FUNCTION_BLOCK "FB_FW_x"   // FB11, STL
TITLE = Fahrwagensteuerung
{ S7_Optimized_Access := 'FALSE' }
AUTHOR : MS
// stored: AutoNumber false
   VAR
      ZST : Struct   // ZUSTAND
         BEREIT : Bool;   // Fahrwagen wartet auf Fahrbefehl
         AKTIV : Bool;   // Fahrwagen bearbeitet Fahrbefehl
         FEHLER : Bool;   // Fahrwagen gestört
         REFERENZIERT : Bool;   // REFERENZIERT
         HEBEN_AKT : Bool;   // Heben aktiv
         SENKEN_AKT : Bool;   // Senken aktiv
         VORWAERTS_AKT : Bool;   // Fahrt zur nächst höheren Position aktiv
         RUECKWAERTS_AKT : Bool;   // Fahrt zur nächst niedrigeren Position aktiv
         Befehl_ok : Bool;   // Befehl angenommen
         Befehl_nok : Bool;   // Befehl abgelehnt
         Befehl_done : Bool;   // Befehl ausgeführt
         Tipp : Bool;   // BA Tippbetrieb interner Zustand
         Hand : Bool;   // BA Handbetrieb interner Zustand
         Auto_Stop : Bool;   // BA Automatikbetrieb angehalten interner Zustand
         Auto : Bool;   // BA Auto interner Zustand
         Semi : Bool;   // Semiautomatik
         POSITION_li : Byte;   // Fahrwagenposition
         Ebene_li : Byte;   // Fahrwagen Hubebene
         PosInc : DInt;   // Position in Inkrementen
         HubInc_li : DInt;   // Hubposition in Inkrementen
         Oben_li : Bool;   // Fahrwagen ist Oben
         Z_Sensor_li : Bool;   // Fahrwagen steht auf Z-Sensor
         Unten_li : Bool;   // Fahrwagen ist Unten
         HubSensor_li : Bool;   // Fahrwagen steht auf Hubsensor
         low_SU_li : Bool;   // niedrigster gültiger SU aktiv
         Mittig : Bool;   // Fahrwagen steht auf Positionsmitte
         HW_mittig : Bool;   // Fahrwagen steht mittig auf Höhenwechsel
         old_vor : Bool;   // letzte Fahrtrichtung war vorwärts
         schieben : Bool;   // FW wird geschoben
         SoftStop : Bool;   // FW wartet auf Freigabe Fahrbereich
         Halt : Bool;   // FW Befehlsabarbeitung angehalten
         Ofs_mittig : Bool;   // FW steht auf Freifahrmitte
         PosStop : Bool;   // Softstop auf Grund gesperrter Position
         schieben_erlaubt : Bool;   // Handbetrieb unterbinden, FW kann noch geschoben werden
         Ofs_Bereich : Bool;   // Tiefsenkbereich
         free : Bool;   // erlaubt die Verwendung durch FB9, bei getakteter Anlage
         POSITION_re : Byte;   // Fahrwagenposition
         Ebene_re : Byte;   // Fahrwagen Hubebene
         Oben_re : Bool;   // Fahrwagen ist Oben
         Z_Sensor_re : Bool;   // Fahrwagen steht auf Z-Sensor
         Unten_re : Bool;   // Fahrwagen ist Unten
         HubSensor_re : Bool;   // Fahrwagen steht auf Hubsensor
         low_SU_re : Bool;   // niedrigster gültiger SU aktiv
         res165 : Bool;
         res166 : Bool;
         res167 : Bool;
         Res_B17 : Byte;   // FEHLER INFORMATION Byte 2
         WT_DB_NR_li : Byte;   // Nr des WT_DB-100
         WT_DB_NR_re : Byte;   // Warenstangen-Nr.
         WT_NR_LANG_li : DWord;   // lange Warenträgernummer für PC
         Befehl_akt : Byte;   // aktueller MicroBefehl
         UP_ON : Bool;   // BEFEHL LÄUFT ALS UNTERPROGRAMM
         next_Step : Bool;   // nächsten MicroBefehl aktivieren
         new_Bef : Bool;   // zeigt den ersten Aufruf des MicroBefehls
         MicM1 : Bool;   // Microbefehlsmerker, wird bei Umschaltung MicroBefehl gelöscht
         MicM2 : Bool;   // Microbefehlsmerker, wird bei Umschaltung MicroBefehl gelöscht
         MicM3 : Bool;   // Microbefehlsmerker, wird bei Umschaltung MicroBefehl gelöscht
         MicM4 : Bool;   // Microbefehlsmerker, wird bei Umschaltung MicroBefehl gelöscht
         Start_UP : Bool;   // Unterprogramm wurde neu gestartet
         Adr_Next_Step : Word;   // Adresse des Bytes mit der abzuarbeitenden Schritt-Nr.
         UP_RET_ADR : Word;   // RÜCKSPRUNG_ADRESSE UNTERPROGRAMM
         BEFEHL : DWord;   // WORD30=KENNUNG,BYTE32=QUELLPOSITION,BYTE33=ZIELPOSITION
         Verweil : DInt;   // Verweilzeit WT am FW
         SchiebeInc : DInt;   // Positionsinkrement auf welches der TW geschoben wird
         Speed_Fahrt : Int;
         Speed_Hub_li : Int;
         Rest_Zeit : DInt;   // Restzeit Umsetzen für Ablaufsteuerung
      END_STRUCT;
      IN : Struct   // EINGANGSSIGNALE
         DIR_VOR : Bool;   // Eingang Fahrt vowärts
         DIR_RCK : Bool;   // Eingang Fahrt rückwärts
         Anf_Hub_li : Bool;   // Anforderung linkes Hubwerk
         Anf_Hub_re : Bool;   // Anforderung rechtes Hubwerk
         DIR_HEB_li : Bool;   // Eingang Heben links
         DIR_SENK_li : Bool;   // Eingang Senken links
         DIR_HEB_re : Bool;   // Eingang Heben rechts
         DIR_SENK_re : Bool;   // Eingang Senken rechts
         Knauf_Auto : Bool;   // Handschalter lokal Hand-Auto
         Aktion : Bool;   // Aktionstaste
         Halt : Bool;   // Halttaste in allen BAs aktiv, mit FW-Bewegungstaste quittierbar
         REP_TASTE : Bool;   // REPERATURTASTE UM ENDSCHALTER ZU BRÜCKEN
         QUITT_ALARM : Bool;   // Eingang Alarme quttieren
         Unten : Bool;   // TW ist ganz unten
         Oben : Bool;   // TW ist ganz oben
         Laser_on : Bool;   // Laser ist eingeschaltet --> Freigabe fahren
         BA_Tipp_ext : Bool;   // externe BA Tipp
         BA_Hand_ext : Bool;   // externe BA Hand global
         BA_Auto_Stop_ext : Bool;   // externe BA Automat anhalten
         BA_Auto_ext : Bool;   // externe BA Automatik
         Unten_li : Bool;   // Sensor unten links
         Oben_li : Bool;   // Sensor oben links
         Unten_re : Bool;   // Sensor unten rechts
         Oben_re : Bool;   // Sensor oben rechts
         FahrBreak_on : Bool;   // Fahrbremse eingefallen im FC SpeedOut verwaltet
         HubBreak_on : Bool;   // Hubbremse eingefallen im FC SpeedOut verwaltet
         Pos_ok : Bool;   // Positionierung abgeschlossen
         Hub_ok_li : Bool;
         Com_Reset : Bool;
         Hub_ok_re : Bool;
         PosGr_min : Bool;   // Minimalgrenze durch Position
         PosGr_max : Bool;   // Maximalgrenze durch Position
         Grenze_min : DInt;   // Grenze des aktuell erlaubten Fahrbereiches min
         Grenze_max : DInt;   // Grenze des aktuell erlaubten Fahrbereiches max
      END_STRUCT;
      ErrIn : Struct   // Fehlermeldungen Eingang
         Alarm : Struct
            NotHalt : Bool;   // NotHalt aktiv alle Fehler ersmal unterdrücken
            PosSys : Bool;   // Fehler Positioniersystem
            HubSys_li : Bool;   // Fehler Hubsystem
            HubSys_re : Bool;   // Fehler Hubsystem
            Hub_nok_links : Bool;   // Hub nicht möglich (FU,MS usw.)
            Hub_nok_rechts : Bool;   // Hub nicht möglich (FU,MS usw.)
            Fahrt_nok : Bool;   // Fahren nicht möglich (FU,MS usw.)
            POS_BELEGT_li : Bool;   // Position mit Warenträger belegt
            POS_BELEGT_re : Bool;   // Position mit Warenträger belegt
            BE_Vor : Bool;   // Bereichsende vorwärts
            BE_Rck : Bool;   // Bereichsende rückwärts
            Koll_LF : Bool;   // Kollision Leerfahrt
            Koll_WF : Bool;   // Kollision Warenfahrt
            AFS_BS : Bool;   // Anfahrschutz Bedienseite
            AFS_WS : Bool;   // Anfahrschutz Wartungsseite
            Gurt_UP_links : Bool;   // GURTENDE OBEN
            Gurt_DN_links : Bool;   // GURTENDE UNTEN
            Gurt_UP_rechts : Bool;   // GURTENDE OBEN
            Gurt_DN_rechts : Bool;   // GURTENDE UNTEN
            Last_UeW_links : Bool;   // Lastüberwachung
            Last_UeW_rechts : Bool;   // Lastüberwachung
            F_Brk_Hub_links : Bool;   // Sicherung Bremse Hub links
            F_Brk_Hub_rechts : Bool;   // Sicherung Bremse Hub rechts
            F_Brk_Fahr : Bool;   // Sicherung Bremse Fahrt
            Gurt_UeL_links : Bool;   // Gurtüberlauf
            Gurt_UeL_rechts : Bool;   // Gurtüberlauf
            Profinet_IO_nok : Bool;   // Profinet nok
            Al_res_8 : Bool;
            AL_res_9 : Bool;
            AL_res_10 : Bool;
            AL_res_11 : Bool;
            AL_res_12 : Bool;
         END_STRUCT;
         Warnung : Struct
            Wrn_Optik_PosSys : Bool;   // Positioniersstem Optik schlecht / Linse putzen
            Wrn_Temp_PosSys : Bool;   // Positioniersystem Temperatur zu hoch
            Wrn_Plaus_PosSys : Bool;   // Positioniersystem Plausibilität
            Wrn_WZ_niO_li_1 : Bool;   // Wägezelle nicht o.k.
            Wrn_WZ_niO_li_2 : Bool;   // Wägezelle nicht o.k.
            Wrn_WZ_niO_li_3 : Bool;   // Wägezelle nicht o.k.
            Wrn_WZ_niO_li_4 : Bool;   // Wägezelle nicht o.k.
            Wrn_WZ_niO_re_1 : Bool;   // Wägezelle nicht o.k.
            Wrn_WZ_niO_re_2 : Bool;   // Wägezelle nicht o.k.
            Wrn_WZ_niO_re_3 : Bool;   // Wägezelle nicht o.k.
            Wrn_WZ_niO_re_4 : Bool;   // Wägezelle nicht o.k.
            Wrn_res_10 : Bool;
            Wrn_res_11 : Bool;
            Wrn_WT_nUmsetzbar : Bool;   // am TW befindlicher Warenträger nicht umsetzbar
            Wrn_Temp_Fahr : Bool;   // Übertemperatur Fahrmotor (führt nach Befehlsende zu Fehler)
            Wrn_Temp_Hub : Bool;   // Übertemperatur Hubmotor (führt nach Befehlsende zu Fehler)
         END_STRUCT;
      END_STRUCT;
      OUT : Struct   // AUSGABESIGNALE (mit * bleiben bei Fehler, auch Not-Aus, an)
         VOR : Bool;   // Ausgang "Vorwärts"
         RUECK : Bool;   // Ausgang "Rückwärts"
         POS_EIL : Bool;   // Ausgang "schnelle Fahrt"
         HEBEN : Bool;   // Ausgang "Heben"
         SENKEN : Bool;   // Ausgang "Senken"
         HUB_EIL_li : Bool;   // Ausgang "schneller Hub"
         HUB_EIL_re : Bool;
         HEBEN_li : Bool;   // Heben links
         HEBEN_re : Bool;   // Heben rechts
         SENKEN_li : Bool;   // Senken links
         SENKEN_re : Bool;   // Senken rechts
         res_3 : Bool;
         res_4 : Bool;
         res_5 : Bool;
         res_6 : Bool;
         res_7 : Bool;
         res_8 : Bool;   // *
         res_9 : Bool;   // *
         TIPP : Bool;   // * Tippbetrieb für externe Funktionen
         Req_Laser : Bool;   // * Anforderung Laserdiode
         no_Brms : Bool;   // * Bremsgeschwind. auslassen
         res_12 : Bool;   // *
         res_13 : Bool;   // *
         res_14 : Bool;   // *
         res_15 : Bool;
         res_16 : Bool;
         res_17 : Bool;
         res_18 : Bool;
         res_19 : Bool;
         res_20 : Bool;
         res_21 : Bool;
         Parken : Bool;   // Parkposition
      END_STRUCT;
      Micro : Struct   // Mikrobefehle
         Adr_UP : Array[1..15] of Word;   // Startadresse einer Microbefehlsprogrammkette
         Liste : Array[0..79] of Byte;   // Frei programmierbare Befehlsliste
      END_STRUCT;
      PAR : Struct   // PARAMETER
         FW_Nr : Byte;   // Fahrwagennummer
         Wichtung : Byte;   // Wichtung des FW bei Schwerpunktberechnung
         TIMER_NR : Int;   // dem FW zugewiesener Timer
         Reihe : Byte;   // Reihe auf der sich FW befindet
         resB : Byte;
         Vorzugsbereich_min : Byte;   // Vorzugsbereich für FB9
         Vorzugsbereich_max : Byte;   // Vorzugsbereich für FB9
         Aktionsbereich_min : Byte;   // Aktionsbereich für FB9
         Aktionsbereich_max : Byte;   // Aktionsbereich für FB9
         resInt : Int;
         Fahrt : Struct
            FAHRBEREICH_MIN : Byte;   // Fahrbereich Anfang
            FAHRBEREICH_MAX : Byte;   // Fahrbereich Ende
            REF_Pos : Byte;   // Referenzposition
            Abstand_vor : DInt;   // min. Abstand zum Nachbar-FW in Vorwärtsrichtung
            dyn_Eil : DInt;
            MessOffset : DInt;   // Offset für PosSystem
            Dir_negativ : Byte;   // Zählrichtung umkehren
            ErrCount : Byte;   // Anzahl der Messversuche bei Fehlmessung
            Bereich_Pos : DInt;   // dieser Bereich gilt als Position mittig
            resD : DInt;
            Bereich_Ziel : DInt;   // Bereich Geschwindigkeit aus
            max_Anhalteweg : DInt;
            Bereich_lngsm : DInt;   // Bereich Geschwindigkeit langsam
            TO_Fahren : S5Time;   // Timeout für Fahrt von Sensor zu Sensor
            Offset_SoftStop : Int;   // Zusätzlicher Abstand bei Softstop
            delta_s : Int;   // Für Timeout Fahren Anzahl der Inkremente, die als Bewegung gelten.
            resT : S5Time;
            WT_Speed : Int;   // Vorgabe in % vom WT (0 == min Speed)
            Park_Pos : Int;   // Parkposition, wenn 5min nichts zu tun
            Count_Park : Int;   // Sollwert Parken nach xxx Sekunden (max.3000)
            Fahr_DBNr : Int;
         END_STRUCT;
         Hub : Struct
            Hub_DBNr : Int;
            WT_Speed : Int;   // Vorgabe vom WT in % (0 = min)
            resInt : Int;
            Dir_negativ_re : Byte;   // Zählrichtung umkehren
            ErrCount_re : Byte;   // Anzahl der Messversuche bei Fehlmessung
            MessOffset_li : DInt;   // Offset für PosSystem
            Dir_negativ_li : Byte;   // Zählrichtung umkehren
            ErrCount_li : Byte;   // Anzahl der Messversuche bei Fehlmessung
            Bereich_Pos : DInt;   // dieser Bereich gilt als Sensor mittig
            resD : DInt;
            Bereich_Ziel : DInt;   // Bereich Geschwindigkeit aus
            MessOffset_re : DInt;   // Offset für PosSystem
            Bereich_lngsm : DInt;   // Bereich Geschwindigkeit langsam
            TO_Heben_Senken_hi : S5Time;   // TimeOUT
            TO_Heben_Senken_low : S5Time;
            delta_s : Int;   // Für Timeout Fahren Anzahl der Inkremente, die als Bewegung gelten.
            TO_HW : S5Time;   // Timeout Höhenwechsel
            TV_HubSensor : S5Time;   // Verzögerung Hubsensor
            Ebene0 : DInt;   // Definition Hub-Sensor an diesem Inkrement
            Ebene1 : DInt;   // niedrigste Ebene=0
            Ebene2 : DInt;   // höchste Ebene=7 bzw. letzte die <>0
            Ebene3 : DInt;
            Ebene4 : DInt;
            Ebene5 : DInt;
            Ebene6 : DInt;
            Ebene7 : DInt;
            SU_Ebenen : Byte;   // jedes Bit aktiviert eine Ebene als SU-Ebene
            Z_Ebene : Byte;   // Nr. der Z-Ebene 0-->keine Z-Ebene
            SO_Ebene : Byte;   // Nr. der SO-Ebene 0-->nicht zulässig
            SUF_Ebene : Byte;   // Nr. der SUF-Ebene 0-->nicht zulässig
         END_STRUCT;
         Free : Struct   // frei verwendbarer Parameterbereich
            TDR_Pause : Int;   // Pausenzeit Trommeldrehen
            TDR_Drehen : Int;   // Drehzeit Trommeldrehen
            Ziel_Inc : DWord;
            resW3 : Word;
            TS_Ablasszeit : Int;   // Zeit für Ablassen Tropfschale
            TS_MV_Zeit : Int;   // Zeit die Ventil zum schließen braucht
            TS_Takte_leeren : Byte;
            TS : Bool;   // Tropfschale vorhanden
            FG_Leeren : Bool;   // Freigabe leeren Tropfschale
            TS_Ablass_Sonderpos : Bool;   // Tropfschale wird nicht auf Posmitte abgelassen --> Sonderbefehl Ablassfahrt
            res153 : Bool;
            res154 : Bool;
            res155 : Bool;
            Z_no_Brms : Bool;   // vor Z keine Bremsgeschwind.
            Laser_req : Bool;
            Laser : DWord;   // Laser-Temp-Daten
         END_STRUCT;
      END_STRUCT;
      TMP : Struct   // HILFSDATEN
         Hub_Ebenen : Byte;   // aktuell gültige Ebenen
         Zielebene_re : Byte;   // aktuell anzufahrende Ebene
         Zielebene_li : Byte;   // aktuell anzufahrende Ebene
         ZielPos : Byte;   // Zielposition die der FW anfahren soll
         HubZielInc_li : DInt;   // Ziel des Hubvorganges in Inkrementen
         FahrZielInc : DInt;   // Ziel des aktuellen Fahrvorganges in Inkrementen
         low_SU_Ebene : Byte;   // unterste gültige SU-Ebene
         ErrCount_Possys : Byte;   // Fehlmessungen Zähler
         FHLR_NR : Int;   // Fehlernummer für Meldeevent
         CouPHub : Int;   // Counter Pendelhübe
         EndZiel : Int;   // Ziel des aktuellen Umsetzvorganges
         count1 : Int;   // Zähler 100ms Takt
         count2 : Int;   // Zähler 100ms Takt
         count3 : Int;   // Zähler 100ms Takt
         count4 : Int;   // Zähler 100ms Takt
         count5 : Int;   // Zähler 100ms Takt
         Verweil : DInt;   // Verweilzeit WT am FW
         Dauer : DInt;   // Zeit in s Leerfahrt, Warenfahrt ohne Pendeln und tropfen
         SoftStopInc : DInt;   // Adresse Softstop bei aktiven Watchspeed
         Opt_Start_Pos : Byte;   // Startposition
         Opt_Ziel_Pos : Byte;   // Zielposition
         Zustand : Byte;   // Reserve für Zustandsmeldungen 44.0Warenfahrt
         Count_TS_leeren : Byte;   // Zähler Tropfschale muß abgelassen werden
         HW_akt_li : Bool;   // Höhenwechsel aktiv
         HW_akt_re : Bool;   // Höhenwechsel aktiv
         FM_F_Taste : Bool;   // Flankenmerker
         res : Bool;
         DKL_Sperre : Bool;   // Deckel muß offen bleiben (FW setz bei Pos_mitte in IstPos, zentrales löschen)
         FM_low_SU_li : Bool;   // Flankenmerker unterster gültiger Sensor
         FW_gestartet : Bool;   // für Transportevent Optimierung
         old_hub : Bool;
         old_vor_hoch : Bool;   // letzte Richtung merken
         old_rueck_runter : Bool;   // letzte Richtung merken
         FM_low_SU_re : Bool;   // Flankenmerker unterster gültiger Sensor
         FP_K_Auto : Bool;   // Flanke Knauf Auto für Reset PC-Control
         FP_K_Auto_int : Bool;   // Flanke Knauf Auto im FB11
         noATZ : Bool;   // Abtropfzeit nicht abarbeiten
         noPend : Bool;   // Pendelzeit nicht abarbeiten
         nextQ_Takt : Bool;   // nächste Quelle reset
         nexQuelle : Word;   // nächste Quelle (Befehl)
         AltPos : DInt;   // letzte Position für Timeout Fahren
         AltHub_li : DInt;   // letzte Hubinc für Timeout Heben
      END_STRUCT;
      MLD : Struct   // Meldungen
         Alarm_HW : Struct
            PosSys : Bool;   // Fehler Positioniersystem
            BE_rck : Bool;   // Bereichsende rückwärts
            BE_vor : Bool;   // Bereichsende vorwärts
            HubSys_li : Bool;   // Fehler Hubsystem
            HubSys_re : Bool;   // Fehler Hubsystem
            GE_oben_li : Bool;   // Gurtende oben
            GE_unten_li : Bool;   // Gurtende unten
            GE_oben_re : Bool;   // Gurtende oben
            GE_unten_re : Bool;   // Gurtende unten
            Koll_LF : Bool;   // Kollision Leerfahrt
            Koll_WF : Bool;   // Kollision Warenfahrt
            Afs_BS : Bool;   // Anfahrschutz Bedienseite
            Afs_WS : Bool;   // Anfahrschutz Wartungsseite
            GurtUeL_li : Bool;   // Gurtüberlauf
            GurtUeL_re : Bool;   // Gurtüberlauf
            St_FU_Fahrt : Bool;   // Störung FU Fahrmotor
            F_Brk_Hub_li : Bool;   // Sicherung Bremse Hub links
            F_Brk_Hub_re : Bool;   // Sicherung Bremse Hub rechts
            F_Brk_Fahr : Bool;   // Sicherung Bremse Fahrt
            St_FU_Hub_li : Bool;   // Störung FU Hubmotor
            St_FU_Hub_re : Bool;   // Störung FU Hubmotor
            Last_UeW_li : Bool;   // Lastüberwachung
            Last_UeW_re : Bool;   // Lastüberwachung
            Temp_Fahrt : Bool;   // Temperatur zu hoch Fahrmotor
            Temp_Hub : Bool;   // Temperatur zu hoch Hub
            Laser_TF : Bool;   // Laser-Entfernungsmesser Temperaturfehler
            Laser_PL : Bool;   // Laser-Entfernungsmesser Plausibilitätsfehler
            Profinet_nok : Bool;   // Profinetmodul keine Rückmeldung
            res_1 : Bool;
            res_2 : Bool;
            res_3 : Bool;
            res_4 : Bool;
         END_STRUCT;
         Alarm_SW : Struct
            Fehler_Quitt : Bool;   // Fehler noch nicht quittiert
            BA_ungueltig : Bool;   // Betriebsart ungültig
            ProgErr : Bool;   // Programmfehler
            nReferenz : Bool;   // nicht referenziert
            NotStop : Bool;   // Not-Stop durch WatchSpeed
            Laser_off : Bool;   // Laser schaltet nicht ein
            TO_Fahrt : Bool;   // Timeout Fahrbewegung
            Auto_SU : Bool;   // Umschaltung auf Automatik in gehobener Stellung
            Auto_WT : Bool;   // Umschaltung auf Automatik und WT noch geladen
            WT_change : Bool;   // Vor ausheben WT entfernt oder getauscht
            Hub_not_mittig_li : Bool;   // Hubbewegung bei Position außermittig
            Hub_nen_li : Bool;   // Hubbewegung nicht erlaubt
            TO_Hub_li : Bool;   // Timeout Hubbewegung
            Senken_WT_li : Bool;   // Bad belegt beim Senken
            Senken_Sperre_li : Bool;   // Bad gesperrt beim Senken
            Heben_WT_li : Bool;   // Bad nicht belegt beim Heben
            SO_fehlt_li : Bool;   // Oben verlassen bei Warenfahrt
            SU_fehlt_li : Bool;   // Unten verlassen bei Leerfahrt
            PosTyp_WT_Typ_li : Bool;   // PosTyp und WT_Typ passen nicht zusammen (Trommel im Gestellbad)
            WTon_bei_SU_li : Bool;   // WT am FW obwohl unten
            TO_Hub_re : Bool;   // Timeout Hubbewegung
            Senken_WT_re : Bool;   // Bad belegt beim Senken
            Senken_Sperre_re : Bool;   // Bad gesperrt beim Senken
            Heben_WT_re : Bool;   // Bad nicht belegt beim Heben
            SO_fehlt_re : Bool;   // Oben verlassen bei Warenfahrt
            SU_fehlt_re : Bool;   // Unten verlassen bei Leerfahrt
            PosTyp_WT_Typ_re : Bool;   // PosTyp und WT_Typ passen nicht zusammen (Trommel im Gestellbad)
            WTon_bei_SU_re : Bool;   // WT am FW obwohl unten
            Hub_not_mittig_re : Bool;   // Hubbewegung bei Position außermittig
            Hub_nen_re : Bool;   // Hubbewegung nicht erlaubt
            ALSW_31 : Bool;
            TO_Befehl : Bool;   // TimeOut Befehlsausführung
         END_STRUCT;
         Warnung : Struct
            Optik_PosSys : Bool;   // Optik schlecht Positioniersystem (Linse putzen)
            Temp_PosSys : Bool;   // Temperatur zu hoch Positioniersystem
            Temp_Fahrt : Bool;   // Temperatur zu hoch Fahrmotor
            Temp_Hub : Bool;   // Temperatur zu hoch Hubmotor
            LSA : Bool;   // Vor-Warnung Laser-Ausfall
            Bh0 : Bool;   // Warnung vorrauss. Lebensdauer erreicht
            Bh100 : Bool;   // Warnung vorrauss. Lebensdauer<100h
            Bh1000 : Bool;   // Warnung vorrauss. Lebensdauer<1000h
            Wrn_Plaus_PosSys : Bool;   // Warnung Plausibilitaet Positioniersystem
            Wrn_WZ_niO_li_1 : Bool;   // Wägezelle nicht o.k.
            Wrn_WZ_niO_li_2 : Bool;   // Wägezelle nicht o.k.
            Wrn_WZ_niO_li_3 : Bool;   // Wägezelle nicht o.k.
            Wrn_WZ_niO_li_4 : Bool;   // Wägezelle nicht o.k.
            Wrn_WZ_niO_re_1 : Bool;   // Wägezelle nicht o.k.
            Wrn_WZ_niO_re_2 : Bool;   // Wägezelle nicht o.k.
            Wrn_WZ_niO_re_3 : Bool;   // Wägezelle nicht o.k.
            Wrn_WZ_niO_re_4 : Bool;   // Wägezelle nicht o.k.
            WARN_18 : Bool;
            WARN_19 : Bool;
            WARN_20 : Bool;
            WARN_21 : Bool;
            WARN_22 : Bool;
            WARN_23 : Bool;
            WARN_24 : Bool;
            WARN_25 : Bool;
            WARN_26 : Bool;
            WARN_27 : Bool;
            WARN_28 : Bool;
            WARN_29 : Bool;
            WARN_30 : Bool;
            WARN_WT_nUms : Bool;   // WT am FW nicht umsetzbar
            WARN_nAuto : Bool;   // TW nicht in Automatik
         END_STRUCT;
         AM_ALHW : DWord;
         AM_ALSW : DWord;
         AM_WARN : DWord;
      END_STRUCT;
      HELP : Struct   // Hilfsvariablen frei verwendbar
         Count_PosSys : Int;   // Verzögerungszähler für Warnmeldungen Positioniersysteme
         Count_Laser_on : Int;
         Count_Parkpos : Int;
         Endziel_WT : Byte;   // Endziel z.Bsp. aus Wtransparenten QT
         QTZiel : Byte;   // QT-Ziel wird an WT-DB kopiert
         Grenze_min : Int;   // für FB9 aktueller Aktionsbereich
         Grenze_max : Int;   // für FB9 aktueller Aktionsbereich
         Speed_Hub_re : Int;
         ResI_8 : Int;
         ResI_9 : Int;
         ResI_10 : Int;
         AuftragWT_li : DInt;   // WT-Nr lang der Auftrag ausgelöst hat.
         AuftragWT_re : DInt;
         HubInc_re : DInt;
         WT_NR_LANG_re : DWord;   // lange Warenträgernummer für PC
         HubZielInc_re : DInt;
         AltHub_re : DInt;   // letzte Hubinc für Timeout Heben
         ResDI_5 : DInt;
         ResDI_6 : DInt;
         ResDI_7 : DInt;
         ResDI_8 : DInt;
         Last_1 : Real;
         Last_2 : Real;
         WZ_links_1 : Real;
         WZ_links_2 : Real;
         WZ_links_3 : Real;
         WZ_links_4 : Real;
         WZ_rechts_1 : Real;
         WZ_rechts_2 : Real;
         WZ_rechts_3 : Real;
         WZ_rechts_4 : Real;
         F_Halt : Bool;   // Flankenmerker
         T_Halt : Bool;   // Taste Halt
         FP_Auto : Bool;   // Flanke Auto
         res_4 : Bool;
         res_5 : Bool;
         res_6 : Bool;
         res_7 : Bool;
         res_8 : Bool;
         res_9 : Bool;
         res_10 : Bool;
         res_11 : Bool;
         res_12 : Bool;
         res_13 : Bool;
         res_14 : Bool;
         res_15 : Bool;
         res_16 : Bool;
         res_17 : Bool;
         res_18 : Bool;
         res_19 : Bool;
         res_20 : Bool;
         res_21 : Bool;
         res_22 : Bool;
         res_23 : Bool;
         res_24 : Bool;
         res_25 : Bool;
         res_26 : Bool;
         res_27 : Bool;
         res_28 : Bool;
         res_29 : Bool;
         res_30 : Bool;
         Last_button_rck : Bool;   // für Handbetrieb letzte Richtungstaste rück
         Last_button_vor : Bool;   // für Handbetrieb letzte Richtungstaste vor
         Tol_UeW_WZ : Real;   // Toleranzwert überwachung Wägezellen
         AW_WZ_li_vorn : Real;
         Sum_WZ_li_vorn : Real;
         AW_WZ_li_hinten : Real;
         Sum_WZ_li_hinten : Real;
         AW_WZ_re_vorn : Real;
         Sum_WZ_re_vorn : Real;
         AW_WZ_re_hinten : Real;
         Sum_WZ_re_hinten : Real;
         Summe_WZ_li : Real;
         AW_Summe_WZ_li : Real;
         Summe_WZ_re : Real;
         AW_Summe_WZ_re : Real;
      END_STRUCT;
   END_VAR
   VAR_TEMP
      WT_DB_NR_li : Word;   // Nr des WT_DB
      HF_DB_NR : Word;   // Hilfsdb-Nr
      WT_DB_NR_re : Word;   // Nr des WT_DB
      Timer0 : Word;   // nicht in Automatik
      Timer1 : Word;   // Timeout Fahren
      Timer2 : Word;   // Timeout Heben
      Timer3 : Word;   // Laser request
      Timer4 : Word;   // FC-Speedout
      Timer5 : Word;   // Verzögerung SU/SO
      Timer6 : Word;   // Simulation SUL
      Timer7 : Word;   // Timeout TS
      Timer8 : Word;   // frei
      Timer9 : Word;   // frei
      count : Int;
      PCount_hi : Int;
      PCount_low : Int;
      t_DINO : Int;
      Adr_IstPos : DWord;
      Adr_UP : DWord;
      Adr_Hub : DWord;
      Adr_Ebene : DWord;
      Param : DWord;
      SoftStopInc : DInt;
      Verweil : DInt;
      Abstand : DInt;   // Hub- und Fahrziel zu Istpos
      End_Ziel_Inc : DInt;
      Z_Inc : DInt;
      KorrPend : Real;
      Korratz : Real;
      Faktor : Real;
      TO_Hub : S5Time;
      Zeit_ms : Time;
      Nummer : USInt;
      inf1 : Byte;
      inf2 : Byte;
      next_WT_for_Pos : Byte;   // nächster in Position angemeldeter WT
      WT_Typ_li : Byte;
      WT_Typ_re : Byte;
      Pos_WT_Typ : Byte;
      WTon_li : Bool;   // WT am FW
      WT_in_Pos_li : Bool;   // in der Position unter dem FW ist ein WT
      WTon_re : Bool;   // WT am FW
      WT_in_Pos_re : Bool;   // in der Position unter dem FW ist ein WT
      C1_rdy : Bool;   // Counter abgelaufen
      C2_rdy : Bool;   // Counter abgelaufen
      C3_rdy : Bool;   // Counter abgelaufen
      C4_rdy : Bool;   // Counter abgelaufen
      C5_rdy : Bool;   // Counter abgelaufen
      F_Taste : Bool;   // Fahrtaste betätigt
      HW_verboten : Bool;   // Höhenwechsel verboten
      lngsm_Fahr : Bool;
      langsam : Bool;
      immer_schnell_li : Bool;
      lngsm_heb_li : Bool;
      lngsm_snk_li : Bool;
      immer_schnell_re : Bool;
      lngsm_heb_re : Bool;
      lngsm_snk_re : Bool;
      Hub_rdy_li : Bool;
      Hub_rdy_re : Bool;
      skip : Bool;   // Überspringen (z.B. nicht anfahrbare Pos)
      noMove : Bool;
      FN_low_SU_li : Bool;
      FN_low_SU_re : Bool;
      "Return" : Bool;   // Rückgabeinformation
      Bef_deleted : Bool;   // Befehl wurde in diesem Zyklus gelöscht
      new : Bool;
      BA_Wxl : Bool;   // Betriebsart gewechselt
      Freigabe : Bool;
      Typ_chk : Bool;   // 0=einfacher Check 10h 20h, 1=detailcheck 11h 12h usw.
      ErrPosSys : Bool;   // Verzögerung PosSys-Warnungen
      chk_WT : Bool;
      Kollision : Bool;   // Auswertung WZ
      WT_151_li : Bool;
      WT_151_re : Bool;
      WT_161_li : Bool;
      WT_161_re : Bool;
   END_VAR
BEGIN

NETWORK
TITLE = Initialisieren und Manipulieren
// Berechnung und Beeinflussung wichtiger Variablen.
//-------------------------
//Timer-Counter-Verwaltung
//-------------------------
      L     #PAR.TIMER_NR;
      T     #Timer0;  //nicht Automatik
      +     1;
      T     #Timer1;  //Timeout Fahren
      +     1;
      T     #Timer2;  //Timeout Heben links
      +     1;
      T     #Timer3;  //Laser ein
      +     1;
      T     #Timer4;  //FC-Speedout
      +     1;
      T     #Timer5;  //Verz. SU/SO
      +     1;
      T     #Timer6;  //Sim SUL
      +     1;
      T     #Timer7;  //Timeout Tropfwanne
      +     1;
      T     #Timer8;  //Timeout Heben rechts
      +     1;
      T     #Timer9;  //frei


//Counter 100ms-Takt
      L     #TMP.count1;  //Timeout Befehl
      L     0;
      <=I;
      =     #C1_rdy;
      L     #TMP.count2;  //Hub erlaubt
      L     0;
      <=I;
      =     #C2_rdy;
      L     #TMP.count3;  //Microbefehl
      L     0;
      <=I;
      =     #C3_rdy;
      L     #TMP.count4;  //Microbefehl
      L     0;
      <=I;
      =     #C4_rdy;
      L     #TMP.count5;  //freie Verwendung
      L     0;
      <=I;
      =     #C5_rdy;

      AN    "Imp_2Hz";  //500ms-Impuls
      ON    "DB_ANLAGE".config.Anl_getaktet;
      JC    free;
      L     0;
      L     #TMP.ZielPos;
      <>I;
      S     #TMP.nextQ_Takt;
      JC    trQ;
      AN    #ZST.BEREIT;
      JC    free;
      A     #TMP.nextQ_Takt;
      R     #TMP.nextQ_Takt;
      JC    free;
      L     0;
trQ:  T     #TMP.nexQuelle;

free: NOP   0;

      AN    "Imp_10Hz";  //100ms-Impuls
      O     #ZST.FEHLER;  //keine Timerbearbeitung im Fehlerzustand
      JC    nImp;

      L     #PAR.Fahrt.Count_Park;
      L     10;
      *I;
      AN    #ZST.BEREIT;
      JC    sPPT;
      L     #HELP.Count_Parkpos;
      L     0;
      <=I;
      JC    sPPT;
      L     #HELP.Count_Parkpos;
      +     -1;
sPPT: T     #HELP.Count_Parkpos;

      L     #HELP.Count_Parkpos;
      L     0;
      <=I;
      A(;
      L     0;
      L     #PAR.Fahrt.Park_Pos;
      <>I;
      );
      =     #OUT.Parken;

      A     #C1_rdy;
      JC    sC1;
      L     #TMP.count1;
      +     -1;
      T     #TMP.count1;

sC1:  A     #C2_rdy;
      JC    sC2;
      L     #TMP.count2;
      +     -1;
      T     #TMP.count2;

sC2:  A     #C3_rdy;
      JC    sC3;
      L     #TMP.count3;
      +     -1;
      T     #TMP.count3;

sC3:  A     #C4_rdy;
      JC    sC4;
      L     #TMP.count4;
      +     -1;
      T     #TMP.count4;

sC4:  A     #C5_rdy;
      JC    nImp;
      L     #TMP.count5;
      +     -1;
      T     #TMP.count5;

//-------------------------
//Temporäre Variablen
//-------------------------
nImp: SET;
      R     #Bef_deleted;
      R     #BA_Wxl;
      R     #OUT.TIPP;
      R     #Kollision;

      A     "DB_ANLAGE".config.TypChckDetail;
      =     #Typ_chk;

      L     100;
      T     #PAR.Fahrt.WT_Speed;
      T     #PAR.Hub.WT_Speed;

      L     #PAR.Hub.Z_Ebene;
      L     0;
      <=I;
      JC    noZE;
      CAC;
      L     4;
      *D;
      L     292;  //"DI_FW_1".PAR.Hub.Ebene0
      +D;
      SLD   3;
      T     #Adr_Hub;
      L     DID [#Adr_Hub];
noZE: T     #Z_Inc;

//-------------------------
//alte Richtung merken
//-------------------------
      A     #OUT.VOR;
      O     #OUT.HEBEN;
      S     #TMP.old_vor_hoch;
      R     #TMP.old_rueck_runter;

      A     #OUT.RUECK;
      O     #OUT.SENKEN;
      R     #TMP.old_vor_hoch;
      S     #TMP.old_rueck_runter;

      A     #OUT.VOR;
      S     #ZST.old_vor;
      A     #OUT.RUECK;
      R     #ZST.old_vor;

      A     #ZST.HEBEN_AKT;
      O     #ZST.SENKEN_AKT;
      =     #TMP.old_hub;

//-------------------------
//Flanke Fahrtaste betätigt
//-------------------------
      A     #IN.DIR_VOR;
      O     #IN.DIR_RCK;
      O     #IN.DIR_HEB_li;
      O     #IN.DIR_SENK_li;
      O     #IN.DIR_HEB_re;
      O     #IN.DIR_SENK_re;
      FP    #TMP.FM_F_Taste;
      =     #F_Taste;

      L     DINO;
      T     #t_DINO;

//-------------------------
//Positioniersystem
//-------------------------
      CALL  "FC_Pos_Erk"
      ( Instanz_DB := #t_DINO
      );

      L     #ZST.POSITION_li;  //nur ungerade werden gezählt
      +     +1;
      T     #ZST.POSITION_re;
//-------------------------
//Hubsystem
//-------------------------
      CALL  "FC_Hub_Erk_li"
      ( Instanz_DB := #t_DINO
      );

      CALL  "FC_Hub_Erk_re"
      ( Instanz_DB := #t_DINO
      );

//-------------------------
// Handbetrieb nicht erlaubt
// FW kann noch geschoben werden
//-------------------------
      L     26;
      SLD   3;
      L     #PAR.Reihe;
      +D;
      LAR1;
      OPN   "DI_FW_MANAGER";
      A     DBX [AR1, P#0.0];
      A     #IN.Knauf_Auto;
      =     #ZST.schieben_erlaubt;

      L     #TMP.nexQuelle;
      L     0;
      <>I;
      A     "DB_ANLAGE".config.Anl_getaktet;
      O     #F_Taste;
      R     #ZST.schieben_erlaubt;

//-------------------------
// Wägezellenwerte Hub
// merken
//-------------------------
      A(;
      A     #ZST.Oben_li;
      AN    #OUT.SENKEN_li;
      O;
      A     #ZST.Unten_li;
      AN    #OUT.HEBEN_li;
      );
      NOT;
      JC    WZre;
      L     #HELP.WZ_links_1;
      L     #HELP.WZ_links_2;
      +R;
      L     #HELP.WZ_links_3;
      +R;
      L     #HELP.WZ_links_4;
      +R;
      T     #HELP.AW_Summe_WZ_li;
WZre: A(;
      A     #ZST.Oben_re;
      AN    #OUT.SENKEN_re;
      O;
      A     #ZST.Unten_re;
      AN    #OUT.HEBEN_re;
      );
      NOT;
      JC    WZ_S;

      L     #HELP.WZ_rechts_1;
      L     #HELP.WZ_rechts_2;
      +R;
      L     #HELP.WZ_rechts_3;
      +R;
      L     #HELP.WZ_rechts_4;
      +R;
      T     #HELP.AW_Summe_WZ_re;

// immer
WZ_S: L     #HELP.WZ_links_1;
      L     #HELP.WZ_links_2;
      +R;
      L     #HELP.WZ_links_3;
      +R;
      L     #HELP.WZ_links_4;
      +R;
      T     #HELP.Summe_WZ_li;

      L     #HELP.WZ_rechts_1;
      L     #HELP.WZ_rechts_2;
      +R;
      L     #HELP.WZ_rechts_3;
      +R;
      L     #HELP.WZ_rechts_4;
      +R;
      T     #HELP.Summe_WZ_re;

//-------------------------
//Positionsadressen für
//indirekte Adressierung
//-------------------------
      L     #ZST.POSITION_li;
      L     "DB_POS".LENG;
      *D;
      L     "DB_POS".Offset;
      +D;
      SLD   3;
      T     #Adr_IstPos;
      LAR1;
      OPN   "DB_POS";
      L     0;
      L     DBB [AR1, P#35.0];
      <>I;
      =     #WT_in_Pos_li;

      L     0;
      L     DBB [AR1, P#135.0];
      <>I;
      =     #WT_in_Pos_re;

//-------------------------
//WT-Information laden
//-------------------------
      L     0;
      L     #ZST.WT_DB_NR_li;
      <I;
      =     #WTon_li;
      JCN   nWTl;
      +     100;
      T     #WT_DB_NR_li;
      OPN   DB [#WT_DB_NR_li];
      L     %DBD6;
      T     #ZST.WT_NR_LANG_li;
      L     %DBB35;  //"DB_WTx".WT_Typ
      T     #WT_Typ_li;
      A     %DBX22.4;  //"DB_WTx".WT_151
      =     #WT_151_li;
      A     %DBX22.5;  //"DB_WTx".WT_161
      =     #WT_161_li;
      JU    WTre;

nWTl: L     0;
      T     #WT_DB_NR_li;
      T     #ZST.WT_DB_NR_li;
      T     #ZST.WT_NR_LANG_li;
      T     #WT_Typ_li;
      SET;
      R     #WT_151_li;
      R     #WT_161_li;

WTre: L     0;
      L     #ZST.WT_DB_NR_re;
      <I;
      =     #WTon_re;
      JCN   nWTr;
      +     100;
      T     #WT_DB_NR_re;

      OPN   DB [#WT_DB_NR_re];
      L     %DBD6;
      T     #HELP.WT_NR_LANG_re;
      L     %DBB35;  //"DB_WTx".WT_Typ
      T     #WT_Typ_re;
      A     %DBX22.4;  //"DB_WTx".WT_151
      =     #WT_151_re;
      A     %DBX22.5;  //"DB_WTx".WT_161
      =     #WT_161_re;
      JU    BA;

nWTr: L     0;
      T     #WT_DB_NR_re;
      T     #ZST.WT_DB_NR_re;
      T     #HELP.WT_NR_LANG_re;
      T     #WT_Typ_re;
      SET;
      R     #WT_151_re;
      R     #WT_161_re;


NETWORK
TITLE = Betriebsart/Fehlerquittung
// Verwaltung der Betriebsarten und Fehlerbehandlung
BA:   NOP   0;
//---------------------
//keine BA-->Fehler
//---------------------
      AN    #IN.BA_Auto_ext;
      AN    #IN.BA_Hand_ext;
      AN    #IN.BA_Tipp_ext;
      AN    #IN.BA_Auto_Stop_ext;  // oben oder unten abgebrochen
      AN    #ErrIn.Alarm.NotHalt;
      =     #MLD.Alarm_SW.BA_ungueltig;
//---------------------
//Auto-->Anhalten
//---------------------
      A     #IN.BA_Auto_ext;
      A     #IN.BA_Auto_Stop_ext;  // oben oder unten abgebrochen
      A     #ZST.Befehl_done;
      R     #ZST.Auto;
      R     #ZST.Tipp;
      S     #ZST.Auto_Stop;
      R     #ZST.Hand;
//---------------------
//-->Auto
//---------------------
      L     #ZST.WT_DB_NR_li;
      L     0;
      <>I;
      O(;
      L     #ZST.WT_DB_NR_re;
      L     0;
      <>I;
      );
      A     #IN.BA_Auto_ext;
      A     #IN.Knauf_Auto;
      AN    #ZST.Auto;
      S     #MLD.Alarm_SW.Auto_WT;

      AN    #ZST.Unten_li;
      ON    #ZST.Unten_re;
      O     #IN.Unten_li;
      O     #IN.Unten_re;
      A     #IN.BA_Auto_ext;
      A     #IN.Knauf_Auto;
      AN    #ZST.Auto;
      S     #MLD.Alarm_SW.Auto_SU;

      AN    #ZST.Auto;
      AN    #MLD.Alarm_SW.Auto_SU;
      AN    #MLD.Alarm_SW.Auto_WT;
      A     #IN.BA_Auto_ext;
      A     #IN.Knauf_Auto;
      AN    #IN.BA_Auto_Stop_ext;
      A     #ZST.Befehl_done;
      S     #ZST.Auto;
      R     #ZST.Tipp;
      R     #ZST.Auto_Stop;
      R     #ZST.Hand;
      S     #BA_Wxl;
      JCN   nEvt;

//---------------------
//-->Hand
//---------------------
nEvt: A     #IN.BA_Auto_ext;
      AN    #IN.Knauf_Auto;
      O     #IN.BA_Hand_ext;
      AN    #ZST.Hand;
      A     #ZST.Befehl_done;
      R     #ZST.Auto;
      R     #ZST.Tipp;
      R     #ZST.Auto_Stop;
      S     #ZST.Hand;
      S     #BA_Wxl;
//---------------------
//-->Tipp
//---------------------
      AN    #ZST.Tipp;
      A     #IN.BA_Tipp_ext;
      A     #ZST.Befehl_done;
      R     #ZST.Auto;
      S     #ZST.Tipp;
      R     #ZST.Auto_Stop;
      R     #ZST.Hand;
      S     #BA_Wxl;
//----------------------
//keine BA --> Tipp
//----------------------
      AN    #ZST.Auto;
      AN    #ZST.Tipp;
      AN    #ZST.Auto_Stop;
      AN    #ZST.Hand;
      S     #ZST.Tipp;
      S     #BA_Wxl;
//---------------------
//FW Stoppen u. Stopp quittieren
//---------------------

//Lösung falls Halt-Taste existiert
//vorherige Variante Löschen und diese aktivieren
      A     #IN.Halt;
      AN    #ZST.Halt;
      S     #ZST.Halt;
      JC    SEv;
      A     #F_Taste;
      A     #ZST.Halt;
      R     #ZST.Halt;
      JC    SEv;
      JU    nSEv;

SEv:  NOP   0;

nSEv: NOP   0;
//-------------------------
//Einrichten/Hand erzwingen
//durch Befehlsabbruch
//-------------------------
      A     #IN.BA_Tipp_ext;
      AN    #ZST.Tipp;
      O(;
      A     #ZST.Unten_li;
      O     #ZST.Oben_li;
      O     #ZST.Unten_re;
      O     #ZST.Oben_re;
      A     #IN.BA_Hand_ext;
      AN    #ZST.Hand;
      );
      AN    #OUT.VOR;
      AN    #OUT.RUECK;
      AN    #OUT.HEBEN_li;
      AN    #OUT.SENKEN_li;
      AN    #OUT.HEBEN_re;
      AN    #OUT.SENKEN_re;
      A     #F_Taste;
      JC    resB;
//---------------------
//Befehl löschen, wenn...
//---------------------
      AN    #IN.Knauf_Auto;
      A     #ZST.Halt;
      A     #ZST.Auto;
      A     #F_Taste;
      JC    resB;

      A     #HELP.T_Halt;
      AN    #ZST.Auto;
      JC    resB;

      A     #ZST.Hand;
      AN    #OUT.VOR;
      AN    #OUT.RUECK;
      AN    #OUT.HEBEN_li;
      AN    #OUT.SENKEN_li;
      AN    #OUT.HEBEN_re;
      AN    #OUT.SENKEN_re;
      A     #F_Taste;
      O     #ZST.Tipp;
      JC    resB;

      A     #IN.QUITT_ALARM;
      O     #F_Taste;
      A     #ZST.Hand;
      A     #ZST.FEHLER;
      JC    resB;
      JU    QErr;

resB: L     0;
      T     #ZST.BEFEHL;
      AN    #ZST.Befehl_done;
      S     #ZST.Befehl_done;
      S     #ZST.Befehl_nok;
      R     #ZST.AKTIV;
      S     #ZST.BEREIT;
      R     #TMP.HW_akt_li;
      S     #Bef_deleted;

//----------------------------
//Fehler-Quittung
//----------------------------
QErr: AN    #ZST.Auto;
      A     #F_Taste;
      O     #IN.QUITT_ALARM;
      A     #ZST.FEHLER;
      AN(;
      A     #ZST.Auto;
      AN    #IN.BA_Auto_ext;
      );
      AN    #ErrIn.Alarm.NotHalt;
      JCN   BA_x;
      R     #ZST.FEHLER;

//:::::::::::::::::::::::::::::::
// Schleife über alle Fehler
//:::::::::::::::::::::::::::::::
      L     418;
      SLD   3;
      LAR1;

      L     1;
reQ:  T     #TMP.FHLR_NR;
      L     96;
      >I;
      JC    QEnd;

      AN    DIX [AR1, P#0.0];
      JC    nxQ;
//:::::::::::::::::::::::::::::::
// Fehler gegangen senden
//:::::::::::::::::::::::::::::::
      L     #TMP.FHLR_NR;
      T     #Nummer;

//:::::::::::::::::::::::::::::::
// nächster Fehler
//:::::::::::::::::::::::::::::::
nxQ:  +AR1  P#0.1;
      L     #TMP.FHLR_NR;
      +     1;
      JU    reQ;

//:::::::::::::::::::::::::::::::
// alle Fehler löschen
//:::::::::::::::::::::::::::::::
QEnd: L     0;
      T     #MLD.AM_ALHW;
      T     #MLD.AM_ALSW;
      T     #MLD.AM_WARN;
      T     %DIW408;
      T     %DID410;  //#MLD.Alarm_SW.xx
      SET;
      R     #MLD.Alarm_HW.Koll_LF;
      R     #MLD.Alarm_HW.Koll_WF;
      R     #ErrIn.Alarm.Last_UeW_links;
      R     #ErrIn.Alarm.Last_UeW_rechts;

BA_x: A     #Bef_deleted;
      JC    Ende;
      A     #ZST.Tipp;
      JC    Tipp;
      A     #ZST.Semi;
      JC    Auto;
      A     #ZST.Hand;
      JC    Hand;
      A     #ZST.Auto;
      JC    Auto;
      JU    doit;

NETWORK
TITLE = Tippbetrieb
Tipp: L     0;
      T     #TMP.EndZiel;

      SET;
      S     #OUT.TIPP;
      R     #OUT.HEBEN_li;
      R     #OUT.HEBEN_re;
      R     #OUT.SENKEN_li;
      R     #OUT.SENKEN_re;
      R     #OUT.VOR;
      R     #OUT.RUECK;
      R     #OUT.SENKEN;
      R     #OUT.HEBEN;

// nur eine Taste erlauben
//     L     %DIB50               // alle Tasten
//      UW    w#16#F3              // Anforderung ausblenden
//      DEC   1
//      L     %DIB50               // alle Tasten
//      UW    w#16#F3              // Anforderung ausblenden
//      UW
//      U <>0

      A     #ErrIn.Alarm.Profinet_IO_nok;
      R     #IN.DIR_RCK;
      R     #IN.DIR_VOR;
      R     #IN.DIR_HEB_re;
      R     #IN.DIR_HEB_li;
      R     #IN.DIR_SENK_re;
      R     #IN.DIR_SENK_li;

      A     #IN.DIR_RCK;
      R     #IN.DIR_VOR;
      A     #IN.DIR_VOR;
      R     #IN.DIR_RCK;

      A     #IN.DIR_HEB_li;
      O     #IN.DIR_HEB_re;
      R     #IN.DIR_SENK_re;
      R     #IN.DIR_SENK_li;

      A     #IN.DIR_SENK_li;
      O     #IN.DIR_SENK_re;
      R     #IN.DIR_HEB_re;
      R     #IN.DIR_HEB_li;

//vorwärts
      AN(;
      A     #ErrIn.Alarm.BE_Vor;
      O     #ErrIn.Alarm.Profinet_IO_nok;
      AN    #IN.REP_TASTE;
      );
      A     #IN.DIR_VOR;
      AN    #OUT.RUECK;
      AN    #OUT.SENKEN;
      AN    #OUT.HEBEN;
      =     #OUT.VOR;
      JC    EndT;

//rückwärts
      AN(;
      A     #ErrIn.Alarm.BE_Rck;
      O     #ErrIn.Alarm.Profinet_IO_nok;
      AN    #IN.REP_TASTE;
      );
      A     #IN.DIR_RCK;
      AN    #OUT.VOR;
      AN    #OUT.SENKEN;
      AN    #OUT.HEBEN;
      =     #OUT.RUECK;
      JC    EndT;


//heben beide Seiten
      AN    #ErrIn.Alarm.Gurt_UP_links;
      AN    #ErrIn.Alarm.Last_UeW_links;
      AN    #ZST.Oben_li;
      AN    #IN.Oben_li;
      AN    #ErrIn.Alarm.Gurt_UP_rechts;
      AN    #ErrIn.Alarm.Last_UeW_rechts;
      AN    #ZST.Oben_re;
      AN    #IN.Oben_re;
      AN    #ErrIn.Alarm.Profinet_IO_nok;
      O     #IN.REP_TASTE;
      A     #IN.DIR_HEB_li;
      A     #IN.DIR_HEB_re;
      =     #OUT.HEBEN_li;
      =     #OUT.HEBEN_re;
      =     #OUT.HEBEN;
      JC    EndT;
//heben
      AN    #ErrIn.Alarm.Gurt_UP_links;
      AN    #ErrIn.Alarm.Last_UeW_links;
      AN    #ZST.Oben_li;
      AN    #IN.Oben_li;
      AN    #ErrIn.Alarm.Profinet_IO_nok;
      O     #IN.REP_TASTE;
      A     #IN.DIR_HEB_li;
      =     #OUT.HEBEN_li;
      =     #OUT.HEBEN;
      JC    EndT;

      AN    #ErrIn.Alarm.Gurt_UP_rechts;
      AN    #ErrIn.Alarm.Last_UeW_rechts;
      AN    #ZST.Oben_re;
      AN    #IN.Oben_re;
      AN    #ErrIn.Alarm.Profinet_IO_nok;
      O     #IN.REP_TASTE;
      A     #IN.DIR_HEB_re;
      =     #OUT.HEBEN_re;
      =     #OUT.HEBEN;
      JC    EndT;


//senken beide Seiten
      AN    #ErrIn.Alarm.Gurt_DN_links;
      AN    #ErrIn.Alarm.Last_UeW_links;
      AN    #ErrIn.Alarm.Gurt_UeL_links;
      AN    #ErrIn.Alarm.Gurt_DN_rechts;
      AN    #ErrIn.Alarm.Last_UeW_rechts;
      AN    #ErrIn.Alarm.Gurt_UeL_rechts;
//      UN    #ZST.low_SU_li
      AN    #IN.Unten_li;
//      UN    #ZST.low_SU_re
      AN    #IN.Unten_re;
      AN    #ErrIn.Alarm.Profinet_IO_nok;
      O     #IN.REP_TASTE;
      A     #IN.DIR_SENK_li;
      A     #IN.DIR_SENK_re;
      =     #OUT.SENKEN_li;
      =     #OUT.SENKEN_re;
      =     #OUT.SENKEN;
      JC    EndT;

//senken
      AN    #ErrIn.Alarm.Gurt_DN_links;
      AN    #ErrIn.Alarm.Last_UeW_links;
      AN    #ErrIn.Alarm.Gurt_UeL_links;
//      UN    #ZST.low_SU_li
      AN    #IN.Unten_li;
      AN    #ErrIn.Alarm.Profinet_IO_nok;
      O     #IN.REP_TASTE;
      A     #IN.DIR_SENK_li;
      =     #OUT.SENKEN_li;
      =     #OUT.SENKEN;
      JC    EndT;

      AN    #ErrIn.Alarm.Gurt_DN_rechts;
      AN    #ErrIn.Alarm.Last_UeW_rechts;
      AN    #ErrIn.Alarm.Gurt_UeL_rechts;
//      UN    #ZST.low_SU_re
      AN    #IN.Unten_re;
      AN    #ErrIn.Alarm.Profinet_IO_nok;
      O     #IN.REP_TASTE;
      A     #IN.DIR_SENK_re;
      =     #OUT.SENKEN_re;
      =     #OUT.SENKEN;
      JC    EndT;

//ZUSTANDSBITS
EndT: CLR;  //U     #IN.Knauf_Auto
      =     #OUT.POS_EIL;

      CLR;
      =     #OUT.HUB_EIL_li;
      =     #OUT.HUB_EIL_re;

      A     #OUT.VOR;
      =     #ZST.VORWAERTS_AKT;
      A     #OUT.RUECK;
      =     #ZST.RUECKWAERTS_AKT;
      A     #OUT.HEBEN;
      =     #ZST.HEBEN_AKT;
      A     #OUT.SENKEN;
      =     #ZST.SENKEN_AKT;

      AN    #ZST.VORWAERTS_AKT;
      AN    #ZST.RUECKWAERTS_AKT;
      AN    #ZST.HEBEN_AKT;
      AN    #ZST.SENKEN_AKT;
      A     #C4_rdy;
      A     #C5_rdy;
      =     #ZST.BEREIT;
      NOT;
      =     #ZST.AKTIV;
      JU    Err;


NETWORK
TITLE = Handbetrieb
Hand: L     0;
      T     #TMP.EndZiel;

      L     #ZST.BEFEHL;
      L     16#0000_0000;
      <>D;
      ON    #ZST.BEREIT;
      JC    EndH;

      A     #ZST.schieben_erlaubt;
      A     #IN.Knauf_Auto;
      JC    EndH;

// Fahren
      A     #IN.DIR_VOR;
      O     #IN.DIR_RCK;
      A     #IN.Aktion;
      JC    FAHR;

//Heben
      A(;
      A     #IN.DIR_HEB_li;
      O     #IN.DIR_SENK_li;
      O     #IN.DIR_HEB_re;
      O     #IN.DIR_SENK_re;
      );
      A     #IN.Aktion;
      JC    HUB;

      JU    Err;  // EndH

HUB:  L     16#F00E_0000;
      T     #ZST.BEFEHL;
      JU    EndH;

FAHR: L     16#F00F_0000;
      T     #ZST.BEFEHL;

EndH: NOP   0;

NETWORK
TITLE = Automatikbetrieb
Auto: A     #ZST.FEHLER;
      JC    ErrA;
//---------------------
//Befehl löschen
//---------------------
      L     #ZST.BEFEHL;
      L     0;
      ==D;
      R     #ZST.UP_ON;
      JC    EndA;
//---------------------
//Prüfung neuer Befehl?
//---------------------
      AN    #ZST.BEREIT;
      JC    doit;
      R     #TMP.noATZ;
      R     #TMP.noPend;

      L     0;
      T     #ZST.Rest_Zeit;

      L     %DIW30;
      L     16#F0F0;
      AW;
      L     16#F000;
      ==I;
      JC    FBok;  //F-Befehl
      JU    flt;
//---------------------
//Befehlsannahme
//---------------------
FBok: L     0;
      L     %DIB32;  //Quellposition im FB?
      ==I;
      JC    ZPOS;
      L     %DIB32;
      L     #PAR.Fahrt.FAHRBEREICH_MIN;
      <I;
      JC    flt;
      L     %DIB32;
      L     #PAR.Fahrt.FAHRBEREICH_MAX;
      >I;
      JC    flt;
ZPOS: L     0;
      L     %DIB33;
      ==I;
      JC    STFB;
      L     %DIB33;
      L     #PAR.Fahrt.FAHRBEREICH_MIN;
      <I;
      JC    flt;
      L     %DIB33;
      L     #PAR.Fahrt.FAHRBEREICH_MAX;
      >I;
      JC    flt;
//Befehl annehmen
STFB: L     0;
      L     %DIB31;
      ==I;
      JC    flt;
      +     -1;
      L     2;
      *D;
      L     72;
      +D;
      SLD   3;
      T     #Adr_UP;  //Adresse der Startadresse des UP
      L     DIW [#Adr_UP];
      T     #ZST.Adr_Next_Step;
      S     #ZST.Befehl_ok;
      S     #ZST.AKTIV;
      S     #ZST.new_Bef;
      S     #ZST.Start_UP;
      R     #ZST.BEREIT;
      R     #ZST.Befehl_done;
      R     #ZST.Befehl_nok;
      R     #ZST.MicM1;
      R     #ZST.MicM2;
      R     #ZST.MicM3;
      R     #ZST.MicM4;
      R     #ZST.free;

      L     %DIB31;  //kein Umsetzbefehl
      L     3;
      <>I;
      JC    doit;

      L     %DIB32;
      T     #inf1;
      L     %DIB33;
      T     #inf2;

      L     #inf2;
      L     0;
      ==I;
      =     #new;

      CALL  "FC_Transzeit"
      ( Pos          := #ZST.POSITION_li,
        Quelle       := #inf1,
        Ziel         := #inf2,
        FW_Nr        := #PAR.FW_Nr,
        ChkLeerfahrt := #new,
        StartPos     := FALSE,
        KorrTime     := DINT#0,
        Fahrzeit     := #ZST.Rest_Zeit
      );

      JU    doit;
flt:  S     #ZST.Befehl_nok;
      L     0;
      T     #ZST.BEFEHL;
      JU    ErrA;

EndA: NOP   0;

NETWORK
TITLE = Befehlsabarbeitung
// Befehlscheck und Ausführung
doit: NOP   0;
      SET;
      R     #lngsm_Fahr;
      R     #langsam;
      R     #OUT.POS_EIL;
      R     #OUT.HUB_EIL_li;
      R     #OUT.HUB_EIL_re;

      L     1.0;
      T     #KorrPend;
      L     0.0;
      T     #Korratz;

      L     0;
      T     #PAR.Free.Ziel_Inc;

      L     #Adr_IstPos;
      LAR1;
      OPN   "DB_POS";
      A     DBX [AR1, P#7.6];  //immer schneller Hub
      =     #immer_schnell_li;

      A     DBX [AR1, P#7.5];  //langsam Heben Badparameter
      =     #lngsm_heb_li;
      A     DBX [AR1, P#7.4];  //langsam Senken Badparameter
      =     #lngsm_snk_li;  //langsam Senken WT-Parameter

      A     DBX [AR1, P#107.6];  //immer schneller Hub
      =     #immer_schnell_re;

      A     DBX [AR1, P#107.5];  //langsam Heben Badparameter
      =     #lngsm_heb_re;
      A     DBX [AR1, P#107.4];  //langsam Senken Badparameter
      =     #lngsm_snk_re;  //langsam Senken WT-Parameter

      AN    #WTon_li;
      JC    WTon_re;

      OPN   DB [#WT_DB_NR_li];
      L     %DBD42;  //Korrekturfaktor Abtropfen
      T     #Korratz;

      A     %DBX22.0;  //langsam senken
      S     #lngsm_snk_li;
      A     %DBX22.1;  //langsam heben
      S     #lngsm_heb_li;
      A     %DBX22.2;  //langsam Fahren
      =     #lngsm_Fahr;

WTon_re:NOP   0;
      AN    #WTon_re;
      JC    strt;

      OPN   DB [#WT_DB_NR_re];
      A     %DBX22.0;  //langsam senken
      S     #lngsm_snk_re;
      A     %DBX22.1;  //langsam heben
      S     #lngsm_heb_re;
      A     %DBX22.2;  //langsam Fahren
      S     #lngsm_Fahr;

      L     #Korratz;
      L     %DBD42;  //Korrekturfaktor Abtropfen
      >R;
      JC    strt;
      T     #Korratz;

strt: L     #ZST.BEFEHL;
      L     0;
      ==D;
      JC    Ende;

      L     DINO;
      T     #t_DINO;

      CALL  "FC_VAR_SPL"
      ( Instanz_DB   := #t_DINO,
        Nr_MicroBef  := #ZST.Befehl_akt,
        next_Step    := #ZST.next_Step,
        Adr_MicroBef := #ZST.Adr_Next_Step
      );

      SET;
      L     #ZST.Befehl_akt;
      JL    list;
      JU    Ende;  //0  Ende UP
      JU    Chk;  //1  Quelle belegt und Ziel frei?
      JU    SetQ;  //2  Quelle als Ziel setzen
      JU    SetZ;  //3  Ziel setzen
      JU    Expo;  //4  Warte bis Expositionszeit abgelaufen
      JU    PosA;  //5  Positionierung Automatik
      JU    PosH;  //6  Positionierung Hand
      JU    HubO;  //7  Heben bis Oben Automatik
      JU    HubZ;  //8  Heben bis Z Automatik
      JU    HubU;  //9  Senken bis Unten Automatik
      JU    HubH;  //10 Heben/Senken Hand
      JU    Pend;  //11 Pendeln
      JU    ATZ;  //12 Abtropfen
      JU    PErr;  //13
      JU    ChkA;  //14 WT-Nr lang,ist die Auftrag augelöst
      JU    PErr;  //15
      JU    PmWT;  //16 Ziel berechnen: Pos.-Mitte WT aufnehemen
      JU    PoWT;  //17 Ziel berechnen: Pos.-Mitte - Offset
      JU    HubF;  //18 Heben bis Leerfahrebene
      JU    PErr;  //19
      JU    WZ_m;  //20 Startwerte Wägezellen merken
      JU    UP01;  //21 Unterprogramm starten
      JU    UP02;  //22 Unterprogramm starten
      JU    UP03;  //23 Unterprogramm starten
      JU    UP04;  //24 Unterprogramm starten
      JU    UP05;  //25 Unterprogramm starten
      JU    UP06;  //26 Unterprogramm starten
      JU    UP07;  //27 Unterprogramm starten
      JU    UP08;  //28 Unterprogramm starten
      JU    UP09;  //29 Unterprogramm starten
      JU    UP10;  //30 Unterprogramm starten
      JU    UP11;  //31 Unterprogramm starten
      JU    UP12;  //32 Unterprogramm starten
      JU    UP13;  //33 Unterprogramm starten
      JU    UP14;  //34 Unterprogramm starten
      JU    UP15;  //35 Unterprogramm starten
list: JU    PErr;

//------------------------------------
//Ende UP
//------------------------------------
Ende: L     0;  //Ausgänge aus
      T     %DIW68;

      A     #Bef_deleted;
      JC    BefD;

      A     #ZST.UP_ON;  //UP läuft?
      JC    REUP;

BefD: AN    "DB_ANLAGE".BA.Automat_ein;
      O     "DB_ANLAGE".config.Anl_getaktet;
      JC    off;

off:  R     #ZST.AKTIV;
      S     #ZST.BEREIT;
      S     #ZST.Befehl_done;
      R     #ZST.Befehl_ok;
      R     #TMP.HW_akt_li;
      R     #TMP.HW_akt_re;
      R     #ZST.SoftStop;
      R     #ZST.RUECKWAERTS_AKT;
      R     #ZST.VORWAERTS_AKT;
      R     #ZST.HEBEN_AKT;
      R     #ZST.SENKEN_AKT;
      R     #IN.Anf_Hub_li;
      R     #IN.Anf_Hub_re;
      R     #ZST.UP_ON;

      L     0;
      T     #TMP.EndZiel;
      T     #ZST.Befehl_akt;
      T     #ZST.Adr_Next_Step;  //Adresse
      T     #ZST.BEFEHL;
      T     #TMP.Opt_Ziel_Pos;
      T     #TMP.ZielPos;
      T     #TMP.Zielebene_li;
      T     #TMP.Zielebene_re;
      T     #TMP.FahrZielInc;
      T     #TMP.HubZielInc_li;
      T     #HELP.HubZielInc_re;
      T     #HELP.AuftragWT_li;
      T     #HELP.AuftragWT_re;
      JU    ErrA;

REUP: R     #ZST.UP_ON;
      S     #ZST.next_Step;
      L     #ZST.UP_RET_ADR;
      T     #ZST.Adr_Next_Step;
      JU    ErrA;

//------------------------------------
//Quelle belegt und Ziel frei?
//------------------------------------
Chk:  AN    #ZST.Auto;
      O     #WTon_li;
      O     #WTon_re;
      S     #ZST.next_Step;
      JC    ErrA;

      L     %DIB32;  //Quelle der Ware
      L     0;
      ==I;
      S     #ZST.Befehl_nok;
      JC    Ende;

      L     %DIB32;  //Quelle der Ware
      L     "DB_POS".LENG;
      *I;
      L     "DB_POS".Offset;
      +I;
      SLD   3;
      LAR1;

      OPN   "DB_POS";
      L     0;
      L     DBB [AR1, P#36.0];  //next WT_DB
      ==I;
      JC    Ende;
      T     #next_WT_for_Pos;
      L     100;
      +I;
      T     #HF_DB_NR;

      OPN   DB [#HF_DB_NR];
      L     %DBB35;  //"DB_WT1".WT_Typ
      T     #WT_Typ_li;

      OPN   "DB_POS";
      A     DBX [AR1, P#7.2];  //Ausfahrsperre
      O     DBX [AR1, P#9.0];  //Ausfahrsperre Freigabe
      A     DBX [AR1, P#96.0];  //Bad belegt
      S     #ZST.Befehl_nok;

      OPN   "DB_POS";
      AN    DBX [AR1, P#96.0];  //Bad belegt
      O     DBX [AR1, P#7.2];  //Ausfahrsperre
      O     DBX [AR1, P#9.0];  //Ausfahrsperre Freigabe
      JC    Ende;

      AN    DBX [AR1, P#96.2];  //Vorruf
      AN    DBX [AR1, P#10.2];  //Expozeit ignorieren
      JC    Ende;

      L     %DIB33;  //Ziel der Ware
      L     0;
      ==I;
      S     #ZST.Befehl_nok;
      JC    Ende;

      L     %DIB32;  //Quelle der Ware
      L     %DIB33;  //Ziel der Ware
      +I;
      L     2;
      MOD;
      A     <>0;
      S     #ZST.Befehl_nok;
      JC    Ende;
// Check Hubwerk
      L     %DIB32;  //Quelle der Ware
      L     2;
      MOD;
      A     ==0;
      R     #IN.Anf_Hub_li;
      =     #IN.Anf_Hub_re;
      JC    ChkZ;
      S     #IN.Anf_Hub_li;

      L     #WT_Typ_li;
      L     "WT_Typ_LS";
      ==I;
      =     #IN.Anf_Hub_re;

ChkZ: L     %DIB33;  //Ziel der Ware
      T     #TMP.EndZiel;
      L     "DB_POS".LENG;
      *I;
      L     "DB_POS".Offset;
      +I;
      SLD   3;
      LAR1;
      L     %DIB32;  //Quelle der Ware
      L     %DIB33;  //Ziel der Ware
      <>I;
      OPN   "DB_POS";
      A(;
      A     DBX [AR1, P#9.1];  //Einfahrsperre Freigabe
      AN    DBX [AR1, P#10.3];  //Einfahrsperre Freigabe ignorieren
      O(;
      A     DBX [AR1, P#96.0];  //Bad belegt
      AN    DBX [AR1, P#6.2];  //"DB_POS".POS[0].Quelle
      );
      );
      O     DBX [AR1, P#7.0];  //Einfahrsperre
      S     #ZST.Befehl_nok;
      JC    Ende;

      L     0;
      L     DBB [AR1, P#36.0];  //Next_WT
      <>I;
      A(;
      L     #next_WT_for_Pos;
      <>I;
      );
      AN    DBX [AR1, P#6.2];  //"DB_POS".POS[0].Quelle
      S     #ZST.Befehl_nok;
      JC    Ende;

      L     DBB [AR1, P#11.0];  // "DB_POS".POS[x].Detailtyp
      T     #Pos_WT_Typ;

      L     #WT_Typ_li;  //Hi-Nibble prüfen vom WT
      AW    16#00F0;
      JZ    hiok;

      L     #Pos_WT_Typ;
      AW    16#00F0;
      JZ    hiok;
      <>I;
      S     #ZST.Befehl_nok;
      JC    Ende;

hiok: AN    #Typ_chk;
      JC    ok;

      L     #WT_Typ_li;  //Lo-Nibble prüfen vom WT
      AW    16#000F;
      JZ    ok;

      L     #Pos_WT_Typ;
      AW    16#000F;
      JZ    ok;
      <>I;
      S     #ZST.Befehl_nok;
      JC    Ende;

ok:   OPN   DB [#HF_DB_NR];
      L     %DBB36;  //WT-Ziel bereits festgelegt
      L     0;
      <>I;
      O     %DBX18.6;  //"DB_WT1".FW_Pos
      JC    Zweg;
      L     0;
      L     %DBB21;  //zu sperrende Ziel-Position
      <>I;
      JC    lok;
      OPN   DB [#HF_DB_NR];
      L     #HELP.Endziel_WT;
      T     %DBB36;  //WT-Ziel
      L     0;  // QT-Ziel
      T     %DBB37;

      JU    Zweg;

lok:  L     "DB_POS".LENG;
      *I;
      L     "DB_POS".Offset;
      +I;
      SLD   3;
      LAR1;
      OPN   "DB_POS";
      L     DBB [AR1, P#36.0];  //Next_WT
      L     0;
      <>I;
      AN    DBX [AR1, P#6.2];  //"DB_POS".POS[0].Quelle
      S     #ZST.Befehl_nok;
      JC    Ende;

      L     %DBB21;
      T     %DBB36;  //WT-Ziel

Zweg: OPN   DB [#HF_DB_NR];
      L     %DIB32;  //Quelle der Ware
      L     2;
      MOD;
      A     <>0;
      L     %DBD6;
      JC    AuftragWT_li;
      T     #HELP.AuftragWT_re;
      L     0;
      T     #HELP.AuftragWT_li;
      JU    next_WT_for_Pos;
AuftragWT_li:NOP   0;
      T     #HELP.AuftragWT_li;
      L     0;
      T     #HELP.AuftragWT_re;
next_WT_for_Pos:NOP   0;
      OPN   "DB_POS";
      L     #next_WT_for_Pos;
      T     DBB [AR1, P#36.0];  //Next_WT
      SET;
      S     #ZST.next_Step;
      JU    ErrA;
//------------------------------------
//WT-Nr lang prüfen ob Auftrag von ihr.
//------------------------------------
ChkA: AN    #ZST.Auto;
      O     #WTon_li;
      O     #WTon_re;
      S     #ZST.next_Step;
      JC    ErrA;

      L     #ZST.POSITION_li;
      L     "DB_POS".LENG;
      *I;
      L     "DB_POS".Offset;
      +I;
      SLD   3;
      LAR1;

      OPN   "DB_POS";
      L     DBD [AR1, P#30.0];  //WT_Nr_lang
      L     #HELP.AuftragWT_li;
      <>D;
      A(;
      L     DINT#0;
      <>D;
      );
      O(;
      L     DBD [AR1, P#130.0];  //WT_Nr_lang
      L     #HELP.AuftragWT_re;
      <>D;
      A(;
      L     DINT#0;
      <>D;
      );
      );
      S     #MLD.Alarm_SW.WT_change;
      S     #Bef_deleted;
      JC    Ende;
      S     #ZST.next_Step;

// Hubwerk bestimmen


      JU    ErrA;

//------------------------------------
//Quelle als Ziel setzen
//------------------------------------
SetQ: L     %DIB32;  //Quelle der Ware
      L     0;
      ==I;
      S     #ZST.Befehl_nok;
      JC    Ende;
      A     #WTon_li;
      S     #ZST.next_Step;
      JC    ErrA;
      L     %DIB32;
      T     #TMP.ZielPos;
      S     #ZST.next_Step;
      JU    ErrA;

//------------------------------------
//Ziel setzen
//------------------------------------
SetZ: L     %DIB33;  //Ziel der Ware
      L     0;
      ==I;
      S     #ZST.Befehl_nok;
      JC    Ende;
      L     %DIB33;
      T     #TMP.ZielPos;
      S     #ZST.next_Step;
      JU    ErrA;

//------------------------------------
//Warte bis Expositionszeit abgelaufen
//------------------------------------
Expo: L     %DIB32;
      L     "DB_POS".LENG;
      *I;
      L     "DB_POS".Offset;
      +I;
      SLD   3;
      LAR1;
      OPN   "DB_POS";
      A     DBX [AR1, P#96.3];  //Expozeit ende(fertig)
      O     DBX [AR1, P#10.2];  //Expoende ignorieren
      ON    DBX [AR1, P#96.0];  //Bad nicht belegt
      ON    #ZST.Auto;
      O     #WTon_li;
      O     #WTon_re;
      S     #ZST.next_Step;
      JU    ErrA;

//------------------------------------
//Positionierung Automatik
//------------------------------------
PosA: L     #TMP.ZielPos;
      L     0;
      ==I;
      S     #ZST.next_Step;
      JC    ErrA;

      A     #TMP.HW_akt_li;
      O     #TMP.HW_akt_re;
      JC    Pos;

      L     %DIW30;
      L     16#FF01;
      ==I;
      L     #ZST.SchiebeInc;
      JC    toPo;

      L     #TMP.ZielPos;
      L     "DB_POS".LENG;
      *I;
      L     "DB_POS".Offset;
      +I;
      SLD   3;
      LAR1;
      OPN   "DB_POS";
      L     DBD [AR1, P#22.0];  //Posmitte
      A     #ZST.Oben_li;
      O     #ZST.Oben_re;
      JC    toPo;
      L     DBD [AR1, P#64.0];  //"DB_POS".POS[x].SonderPos_Offset
      -D;
toPo: T     #TMP.FahrZielInc;  //Zielposition in Inkrementen

//Test auf Höhenwechsel
      CALL  "FC_Search_HW"
      ( SO_li           := #ZST.Oben_li,
        SO_re           := #ZST.Oben_re,
        IstPos          := #ZST.PosInc,
        ZielPos         := #TMP.FahrZielInc,
        Bereich_Ziel    := #PAR.Fahrt.Bereich_Pos,
        Bereich_langsam := #PAR.Fahrt.Bereich_lngsm,
        FW_Ebene_li     := #ZST.Ebene_li,
        Zielebene_li    := #TMP.Zielebene_li,
        HW_akt_li       := #TMP.HW_akt_li,
        FW_Ebene_re     := #ZST.Ebene_re,
        Zielebene_re    := #TMP.Zielebene_re,
        HW_akt_re       := #TMP.HW_akt_re
      );

      JU    Pos;

//------------------------------------
// Pos. zur WT-Aufnahme
//------------------------------------
PmWT: L     #Adr_IstPos;
      LAR1;
      OPN   "DB_POS";
      L     DBD [AR1, P#22.0];  //Posmitte
      T     #TMP.FahrZielInc;  //Zielposition in Inkrementen
      JU    Pos;

//------------------------------------
// Pos. zur WT-Freigabe
//------------------------------------
PoWT: L     #Adr_IstPos;
      LAR1;
      OPN   "DB_POS";
      L     DBD [AR1, P#22.0];  //Posmitte
      L     DBD [AR1, P#64.0];  //"DB_POS".POS[x].SonderPos_Offset
      -D;
      T     #TMP.FahrZielInc;  //Zielposition in Inkrementen
      JU    Pos;

//------------------------------------
//Positionierung Hand
//------------------------------------
PosH: AN    #IN.Aktion;
      O;
      AN    #IN.DIR_VOR;
      AN    #IN.DIR_RCK;
      A     #ZST.new_Bef;
      O;
      A     #IN.DIR_VOR;
      A     #IN.DIR_RCK;
      A     #ZST.new_Bef;
      R     #OUT.RUECK;
      R     #OUT.VOR;
      S     #ZST.next_Step;
      JC    ErrA;

      A     #ZST.new_Bef;
      R     #HELP.Last_button_vor;
      R     #HELP.Last_button_rck;

//Richtungswechsel bzw. Taste losgelassen
      A     #IN.DIR_VOR;
      A     #IN.DIR_RCK;
      O(;
      A     #IN.DIR_VOR;
      A     #OUT.RUECK;
      );
      O(;
      A     #IN.DIR_RCK;
      A     #OUT.VOR;
      );
      O(;
      A     #OUT.VOR;
      O     #OUT.RUECK;
      AN    #IN.DIR_VOR;
      AN    #IN.DIR_RCK;
      );
      JC    Such;

//Taste ist gedrückt
      S     #ZST.MicM2;  //merken Taste

      A     #IN.DIR_VOR;
      S     #HELP.Last_button_vor;
      R     #HELP.Last_button_rck;
      A     #IN.DIR_RCK;
      R     #HELP.Last_button_vor;
      S     #HELP.Last_button_rck;

      AN    #HELP.Last_button_vor;
      AN    #HELP.Last_button_rck;
      S     #ZST.next_Step;
      JC    ErrA;

      CALL  "FC_Suche_next_HaltePos"
      ( IstPosInc := #ZST.PosInc,
        Halteweg  := #PAR.Fahrt.max_Anhalteweg,
        vor       := #HELP.Last_button_vor,
        SO_li     := #ZST.Oben_li,
        SO_re     := #ZST.Oben_re,
        ZielPos   := #TMP.ZielPos
      );

      L     #TMP.ZielPos;
      L     #ZST.POSITION_li;
      <I;
      A     #HELP.Last_button_vor;
      S     #ZST.next_Step;
      JC    ErrA;

      L     #TMP.ZielPos;
      L     #ZST.POSITION_li;
      >I;
      A     #HELP.Last_button_rck;
      S     #ZST.next_Step;
      JC    ErrA;
      JU    POut;


Such: AN    #ZST.MicM2;
      JC    HWCk;
      R     #ZST.MicM2;

      AN    #HELP.Last_button_vor;
      AN    #HELP.Last_button_rck;
      S     #ZST.next_Step;
      JC    ErrA;

      CALL  "FC_Suche_next_HaltePos"
      ( IstPosInc := #ZST.PosInc,
        Halteweg  := #PAR.Fahrt.Bereich_lngsm,
        vor       := #HELP.Last_button_vor,
        SO_li     := #ZST.Oben_li,
        SO_re     := #ZST.Oben_re,
        ZielPos   := #TMP.ZielPos
      );

      L     #TMP.ZielPos;
      L     #ZST.POSITION_li;
      <I;
      A     #HELP.Last_button_vor;
      S     #ZST.next_Step;
      JC    ErrA;

      L     #TMP.ZielPos;
      L     #ZST.POSITION_li;
      >I;
      A     #HELP.Last_button_rck;
      S     #ZST.next_Step;
      JC    ErrA;

      L     #TMP.ZielPos;
      L     #ZST.POSITION_li;
      <>I;
      JC    POut;
      L     "DB_POS".LENG;
      *I;
      L     "DB_POS".Offset;
      +I;
      SLD   3;
      LAR1;
      OPN   "DB_POS";
      L     DBD [AR1, P#22.0];  //Posmitte
      A     #ZST.Oben_li;
      O     #ZST.Oben_re;
      JC    nOfs;
      L     DBD [AR1, P#64.0];  //"DB_POS".POS[0].SonderPos_Offset
      -D;
nOfs: L     #ZST.PosInc;
      -D;
      DTR;
      ABS;
      RND;
      L     #PAR.Fahrt.Bereich_Pos;
      >D;
      JC    POut;
      L     #TMP.ZielPos;
      +     2;
      A     #OUT.VOR;
      JC    TPos;
      L     #TMP.ZielPos;
      +     -2;
      A     #OUT.RUECK;
      JC    TPos;
      JU    POut;

TPos: L     #PAR.Fahrt.FAHRBEREICH_MIN;
      <I;
      JC    KorF;
      CAC;
      L     #PAR.Fahrt.FAHRBEREICH_MAX;
      DEC   1;  // HCA: nur ungerade zählen
      >I;
      JC    KorF;
      CAC;
KorF: T     #TMP.ZielPos;

POut: AN    #ZST.Ofs_Bereich;
      JC    PZiel;

      L     #ZST.POSITION_li;
      T     #TMP.ZielPos;

//zur WT-Aufnahme
      A     #IN.DIR_VOR;
      L     #Adr_IstPos;
      LAR1;
      OPN   "DB_POS";
      L     DBD [AR1, P#22.0];  //Posmitte
      JC    SInc;

//Freifahren
      A     #IN.DIR_RCK;
      L     DBD [AR1, P#22.0];  //Posmitte
      L     DBD [AR1, P#64.0];  //"DB_POS".POS[x].SonderPos_Offset
      -D;
      JC    SInc;
      JU    HWCk;

PZiel:L     #TMP.ZielPos;
      L     "DB_POS".LENG;
      *I;
      L     "DB_POS".Offset;
      +I;
      SLD   3;
      LAR1;
      OPN   "DB_POS";
//mit Ware
      L     DBD [AR1, P#22.0];  //Posmitte
      A     #ZST.Oben_li;
      O     #ZST.Oben_re;
      JC    SInc;
//leer
      L     DBD [AR1, P#64.0];  //"DB_POS".POS[x].SonderPos_Offset
      -D;

SInc: T     #TMP.FahrZielInc;


HWCk: CALL  "FC_Search_HW"
      ( SO_li           := #ZST.Oben_li,
        SO_re           := #ZST.Oben_re,
        IstPos          := #ZST.PosInc,
        ZielPos         := #TMP.FahrZielInc,
        Bereich_Ziel    := #PAR.Fahrt.Bereich_Pos,
        Bereich_langsam := #PAR.Fahrt.Bereich_lngsm,
        FW_Ebene_li     := #ZST.Ebene_li,
        Zielebene_li    := #TMP.Zielebene_li,
        HW_akt_li       := #TMP.HW_akt_li,
        FW_Ebene_re     := #ZST.Ebene_re,
        Zielebene_re    := #TMP.Zielebene_re,
        HW_akt_re       := #TMP.HW_akt_re
      );
      SET;
      R     #TMP.HW_akt_li;
      R     #TMP.HW_akt_re;

      JU    Pos;
//------------------------------------
//Heben/Senken Automatik
//------------------------------------
HubZ: L     0;
      L     #PAR.Hub.Z_Ebene;
      ==I;
      S     #MLD.Alarm_SW.ProgErr;
      JC    ErrA;

      L     #TMP.low_SU_Ebene;
      L     #PAR.Hub.Z_Ebene;
      >I;
      S     #MLD.Alarm_SW.ProgErr;
      JC    ErrA;

      L     #ZST.Ebene_li;
      L     #PAR.Hub.Z_Ebene;
      >I;
      S     #ZST.next_Step;
      R     #OUT.HEBEN;
      R     #OUT.SENKEN;
      JC    ErrA;
      JU    HubG;

HubO: L     0;
      L     #PAR.Hub.SO_Ebene;
      ==I;
      S     #MLD.Alarm_SW.ProgErr;
      JC    ErrA;
      JU    HubG;

HubF: L     0;
      L     #PAR.Hub.SUF_Ebene;
      ==I;
      S     #MLD.Alarm_SW.ProgErr;
      JC    ErrA;
      JU    HubG;

HubU: L     #TMP.low_SU_Ebene;
      JU    HubG;

HubG: T     #TMP.Zielebene_li;
      T     #TMP.Zielebene_re;
      L     4;
      *D;
      L     292;  //"DI_FW_1".PAR.Hub.Ebene0
      +D;
      SLD   3;
      T     #Adr_Hub;
      L     DID [#Adr_Hub];
      T     #TMP.HubZielInc_li;
      T     #HELP.HubZielInc_re;
      JU    Hub_Mig;
//------------------------------------
//Heben/Senken Hand
//------------------------------------
HubH: AN    #IN.Aktion;
Hoff: R     #OUT.HEBEN;
      R     #OUT.SENKEN;
      R     #OUT.HEBEN_li;
      R     #OUT.HEBEN_re;
      R     #OUT.SENKEN_li;
      R     #OUT.SENKEN_re;
      R     #IN.Anf_Hub_li;
      R     #IN.Anf_Hub_re;
      S     #ZST.next_Step;
      JC    ErrA;

      AN    #ZST.HW_mittig;
      AN    #ZST.Ofs_mittig;
      =     #HW_verboten;

      A(;
      A     #IN.DIR_HEB_li;
      A     #F_Taste;
      AN    #ZST.Oben_li;
      O;
      A     #IN.DIR_HEB_re;
      A     #F_Taste;
      AN    #ZST.Oben_re;
      );
      AN    #OUT.SENKEN;
      JC    H_UP;

      A(;
      A     #IN.DIR_SENK_li;
      AN    #ZST.low_SU_li;
      O;
      A     #IN.DIR_SENK_re;
      AN    #ZST.low_SU_re;
      );
      AN    #OUT.HEBEN;
      JC    H_DN;

      AN    #OUT.HEBEN;
      AN    #OUT.SENKEN;
      A     #ZST.new_Bef;
      JC    Hoff;
      JU    HW;

//Höhenwechselbehandlung
H_UP: L     0;
      L     #ZST.WT_DB_NR_li;
      <>I;
      A(;
      L     #ZST.WT_DB_NR_re;
      ==I;
      );
      A(;
      AN    #IN.DIR_HEB_li;
      ON    #IN.DIR_HEB_re;
      );
      A     #ZST.Mittig;
      JC    Hoff;

      L     #Adr_IstPos;
      LAR1;
      OPN   "DB_POS";
      L     0;
      L     DBB [AR1, P#36.0];  //Next_WT
      <>I;
      A(;
      L     DBB [AR1, P#136.0];  //Next_WT
      ==I;
      );
      A(;
      AN    #IN.DIR_HEB_li;
      ON    #IN.DIR_HEB_re;
      );
      A     #ZST.Mittig;
      A(;
      A     #ZST.low_SU_li;
      O     #ZST.low_SU_re;
      );
      JC    Hoff;

      L     #Adr_IstPos;
      LAR1;
      OPN   "DB_POS";
      L     0;
      L     DBB [AR1, P#36.0];  //Next_WT
      <>I;
      A(;
      L     DBB [AR1, P#136.0];  //Next_WT
      ==I;
      );
      A     #IN.DIR_HEB_li;
      A     #IN.DIR_HEB_re;
      A     #ZST.Mittig;
      A(;
      A     #ZST.low_SU_li;
      X     #ZST.low_SU_re;
      );
      JC    Hoff;

      AN    #IN.DIR_HEB_li;
      O     #ZST.Oben_li;
      JC    H_UP_re;
      S     #IN.Anf_Hub_li;

      A     #HW_verboten;
      JC    HWT_li;

      L     #ZST.Ebene_li;
      A     #ZST.HubSensor_li;
      JC    HSon_li;  //FW befindet sich auf Ebenenmitte
      L     4;
      *D;
      L     292;  //"DI_FW_1".PAR.Hub.Ebene0
      +D;
      SLD   3;
      T     #Adr_Hub;
      L     #ZST.HubInc_li;  //Istposition Hubbalken in Inkrementen
      L     DID [#Adr_Hub];  //Posmitte der aktuellen Ebene in Inkrementen
      <D;  //FW hat Ebenenmitte dieser Ebene noch vor sich
      L     #ZST.Ebene_li;
      JC    retE_li;  //Suche ab Ist-Ebene beginnen
HSon_li:+     1;  //Suche bei Ist-Ebene+1 beginnen
retE_li:T     #count;  //Suchschleife nach nächster gültigen Ebene
      L     7;
      >=I;
      JC    nZ_li;  //Oberste definierbare Ebene --> Abbruch
      L     #count;  //Ebenenzähler
      +     1;
      L     #TMP.Hub_Ebenen;
      SRW;  //ist das Ebenenbit==TRUE --> A1-Bit==TRUE
      JP    HEf_li;  //Springt, wenn A1-Bit==TRUE (gültige Ebene)
      L     #count;
      +     1;
      JU    retE_li;  //nächste Ebene prüfen

//Höhenwechselebene gefunden
HEf_li:L     #count;  //kann auch Z- bzw. SO-Ebene sein
      T     #TMP.Zielebene_li;
      JU    H_UP_re;

HWT_li:L     0;
      L     #PAR.Hub.Z_Ebene;
      ==I;
      O     #immer_schnell_li;
      JC    nZ_li;
      L     4;
      *D;
      L     292;  //"DI_FW_1".PAR.Hub.Ebene0
      +D;
      SLD   3;
      T     #Adr_Hub;
      L     #ZST.HubInc_li;
      L     DID [#Adr_Hub];
      >I;
      O     #ZST.Z_Sensor_li;
      JC    nZ_li;
      L     #PAR.Hub.Z_Ebene;
      T     #TMP.Zielebene_li;
      JU    H_UP_re;

nZ_li:L     0;
      L     #PAR.Hub.SO_Ebene;
      ==I;
      S     #MLD.Alarm_SW.ProgErr;
      JC    ErrA;
      T     #TMP.Zielebene_li;
      JU    H_UP_re;

H_UP_re:NOP   0;
      AN    #IN.DIR_HEB_re;
      O     #ZST.Oben_re;
      JC    HW;
      S     #IN.Anf_Hub_re;

      A     #HW_verboten;
      JC    HWT_re;

      L     #ZST.Ebene_re;
      A     #ZST.HubSensor_re;
      JC    HSon_re;  //FW befindet sich auf Ebenenmitte
      L     4;
      *D;
      L     292;  //"DI_FW_1".PAR.Hub.Ebene0
      +D;
      SLD   3;
      T     #Adr_Hub;
      L     #HELP.HubInc_re;  //Istposition Hubbalken in Inkrementen
      L     DID [#Adr_Hub];  //Posmitte der aktuellen Ebene in Inkrementen
      <D;  //FW hat Ebenenmitte dieser Ebene noch vor sich
      L     #ZST.Ebene_re;
      JC    retE_re;  //Suche ab Ist-Ebene beginnen
HSon_re:+     1;  //Suche bei Ist-Ebene+1 beginnen
retE_re:T     #count;  //Suchschleife nach nächster gültigen Ebene
      L     7;
      >=I;
      JC    nZ_re;  //Oberste definierbare Ebene --> Abbruch
      L     #count;  //Ebenenzähler
      +     1;
      L     #TMP.Hub_Ebenen;
      SRW;  //ist das Ebenenbit==TRUE --> A1-Bit==TRUE
      JP    HEf_re;  //Springt, wenn A1-Bit==TRUE (gültige Ebene)
      L     #count;
      +     1;
      JU    retE_re;  //nächste Ebene prüfen

//Höhenwechselebene gefunden
HEf_re:L     #count;  //kann auch Z- bzw. SO-Ebene sein
      T     #TMP.Zielebene_re;
      JU    HW;

HWT_re:L     0;
      L     #PAR.Hub.Z_Ebene;
      ==I;
      O     #immer_schnell_re;
      JC    nZ_re;
      L     4;
      *D;
      L     292;  //"DI_FW_1".PAR.Hub.Ebene0
      +D;
      SLD   3;
      T     #Adr_Hub;
      L     #HELP.HubInc_re;
      L     DID [#Adr_Hub];
      >I;
      O     #ZST.Z_Sensor_re;
      JC    nZ_re;
      L     #PAR.Hub.Z_Ebene;
      T     #TMP.Zielebene_re;
      JU    HW;

nZ_re:L     0;
      L     #PAR.Hub.SO_Ebene;
      ==I;
      S     #MLD.Alarm_SW.ProgErr;
      JC    ErrA;
      T     #TMP.Zielebene_re;
      JU    HW;

H_DN: L     0;
      L     #ZST.WT_DB_NR_li;
      <>I;
      A(;
      L     #ZST.WT_DB_NR_re;
      ==I;
      );
      A(;
      AN    #IN.DIR_SENK_li;
      ON    #IN.DIR_SENK_re;
      );
      A     #ZST.Mittig;
      JC    Hoff;

      A     #IN.DIR_SENK_li;
      AN    #ZST.low_SU_li;
      S     #IN.Anf_Hub_li;

      A     #IN.DIR_SENK_re;
      AN    #ZST.low_SU_re;
      S     #IN.Anf_Hub_re;

      L     #TMP.low_SU_Ebene;
      T     #TMP.Zielebene_li;
      T     #TMP.Zielebene_re;
      JU    HW;

//----------------------------------
//Höhenwechselvorgang
//----------------------------------
HW:   L     #TMP.Zielebene_li;
      L     4;
      *D;
      L     292;  //"DI_FW_1".PAR.Hub.Ebene0
      +D;
      SLD   3;
      T     #Adr_Hub;
      L     DID [#Adr_Hub];
      T     #TMP.HubZielInc_li;

      L     #TMP.Zielebene_re;
      L     4;
      *D;
      L     292;  //"DI_FW_1".PAR.Hub.Ebene0
      +D;
      SLD   3;
      T     #Adr_Hub;
      L     DID [#Adr_Hub];
      T     #HELP.HubZielInc_re;
      JU    Hub_Mig;
//------------------------------------
//Pendeln
//------------------------------------
Pend: A     #C3_rdy;
      AN    #ZST.new_Bef;
      O     #TMP.noPend;
      S     #ZST.next_Step;
      JC    ErrA;

      AN    #ZST.new_Bef;
      JC    ErrA;

      L     #Adr_IstPos;
      LAR1;
      OPN   "DB_POS";
      L     DBW [AR1, P#82.0];  //Pendelzeit
      DTR;
      L     #KorrPend;
      *R;
      RND;
      L     0;
      <I;
      S     #ZST.next_Step;
      JC    ErrA;
      CAC;
      L     10;
      *D;
      T     #TMP.count3;
      JU    ErrA;

//------------------------------------
//Abtropfen
//------------------------------------
ATZ:  L     %DIB32;
      L     %DIB33;
      ==I;
      O     #ZST.Z_Sensor_li;
      O     #ZST.Z_Sensor_re;
      S     #ZST.next_Step;
      R     #TMP.DKL_Sperre;
      JC    ErrA;

      A     #C3_rdy;
      AN    #ZST.new_Bef;
      O;
      A     #immer_schnell_li;
      A     #immer_schnell_re;
      S     #ZST.next_Step;
      R     #TMP.DKL_Sperre;
      JC    ErrA;

      AN    #ZST.new_Bef;
      JC    EATZ;
      S     #TMP.DKL_Sperre;

      L     #Adr_IstPos;
      LAR1;
      OPN   "DB_POS";
      L     DBW [AR1, P#84.0];  //Abtropfzeit
      DTR;
      L     #Korratz;
      *R;
      RND;
      L     10;
      *D;
      T     #TMP.count3;
EATZ: JU    ErrA;

//------------------------------------
//Startwerte Wägezellen merken
//------------------------------------
WZ_m: A     #C3_rdy;  // 500 ms warten
      AN    #ZST.new_Bef;
      JC    WZm1;

      AN    #ZST.new_Bef;
      JC    ErrA;

      L     5;
      T     #TMP.count3;
      JU    ErrA;

WZm1: L     #HELP.WZ_links_1;
      L     #HELP.WZ_links_2;
      +R;
      T     #HELP.AW_WZ_li_vorn;

      L     #HELP.WZ_links_3;
      L     #HELP.WZ_links_4;
      +R;
      T     #HELP.AW_WZ_li_hinten;

      L     #HELP.WZ_rechts_1;
      L     #HELP.WZ_rechts_2;
      +R;
      T     #HELP.AW_WZ_re_vorn;

      L     #HELP.WZ_rechts_3;
      L     #HELP.WZ_rechts_4;
      +R;
      T     #HELP.AW_WZ_re_hinten;

      SET;
      S     #ZST.next_Step;
      JU    ErrA;

//------------------------------------
//Unterprogramm starten
//------------------------------------
UP01: L     0;
      JU    UP;
UP02: L     1;
      JU    UP;
UP03: L     2;
      JU    UP;
UP04: L     3;
      JU    UP;
UP05: L     4;
      JU    UP;
UP06: L     5;
      JU    UP;
UP07: L     6;
      JU    UP;
UP08: L     7;
      JU    UP;
UP09: L     8;
      JU    UP;
UP10: L     9;
      JU    UP;
UP11: L     10;
      JU    UP;
UP12: L     11;
      JU    UP;
UP13: L     12;
      JU    UP;
UP14: L     13;
      JU    UP;
UP15: L     14;
      JU    UP;

UP:   L     2;
      *D;
      T     #Adr_UP;
      SET;
      S     #ZST.UP_ON;
      S     #ZST.Start_UP;

      L     #ZST.Adr_Next_Step;
      T     #ZST.UP_RET_ADR;

      L     #Adr_UP;
      L     72;
      +D;
      SLD   3;
      T     #Adr_UP;  //Adresse der Startadresse des UP
      L     DIW [#Adr_UP];
      T     #ZST.Adr_Next_Step;

      L     0;  //Ausgänge aus
      T     %DIB68;
      JU    ErrA;

//------------------------------------
//ungültige Sprungadresse
//------------------------------------
PErr: S     #MLD.Alarm_SW.ProgErr;
      JU    Ende;


NETWORK
TITLE = Positionierung
Pos:  NOP   0;
//------------------------------------
//Positioniervorgang
//------------------------------------
      AN    #IN.Laser_on;
      AN    #ZST.MicM3;
      JC    ErrA;
      S     #ZST.MicM3;

      L     #TMP.FahrZielInc;
      T     #End_Ziel_Inc;

//-------------------
      L     #TMP.FahrZielInc;
      L     #ZST.PosInc;
      -D;
      DTR;
      ABS;
      RND;
      T     #Abstand;

      L     #Abstand;
      L     #PAR.Fahrt.Bereich_Pos;
      <=D;
      A     #ZST.MicM1;  //neuer Befehl noch keine Richtung gewählt
      JC    WSpd;

      L     #TMP.FahrZielInc;
      L     #ZST.PosInc;
      <D;
      S     #OUT.RUECK;
      R     #OUT.VOR;
      S     #ZST.RUECKWAERTS_AKT;
      R     #ZST.VORWAERTS_AKT;
      >D;
      R     #OUT.RUECK;
      S     #OUT.VOR;
      R     #ZST.RUECKWAERTS_AKT;
      S     #ZST.VORWAERTS_AKT;

WSpd: NOP   0;

//-------------------

      CALL  "FC_WATCH_SPEED"
      ( Instanz_DB     := #t_DINO,
        PosInc         := #ZST.PosInc,
        ZielInc        := #TMP.FahrZielInc,
        Grenze_min     := #IN.Grenze_min,
        Grenze_max     := #IN.Grenze_max,
        Bereich_lngsm  := #PAR.Fahrt.Bereich_lngsm,
        Bereich_Pos    := #PAR.Fahrt.Bereich_Pos,
        Dyn_Eil        := #PAR.Fahrt.dyn_Eil,
        Offset         := #PAR.Fahrt.Offset_SoftStop,
        PosGr_min      := #IN.PosGr_min,
        PosGr_max      := #IN.PosGr_max,
        PosStop        := #ZST.PosStop,
        NOTSTOP        := #MLD.Alarm_SW.NotStop,
        Vorwaerts      := #OUT.VOR,
        Rueckwaerts    := #OUT.RUECK,
        SoftStop_aktiv := #ZST.SoftStop,
        ADR_SFT_STOP   := #TMP.SoftStopInc
      );  //Suche nach Hindernissen und evtl. Korrektur des Ziels

      AN    #ZST.SoftStop;
      JC    nSFT;
      R     #TMP.HW_akt_li;
      R     #TMP.HW_akt_re;

      L     #TMP.SoftStopInc;
      T     #TMP.FahrZielInc;

nSFT: L     #TMP.FahrZielInc;
      L     #ZST.PosInc;
      -D;
      DTR;
      ABS;
      RND;
      T     #Abstand;

//Bremsvorgang
      AN    #lngsm_Fahr;
      A     #ZST.Auto;
      =     #OUT.POS_EIL;

      L     #Abstand;
      L     #PAR.Fahrt.Bereich_Pos;
      <=D;
      A     #IN.Pos_ok;
      R     #OUT.VOR;
      R     #OUT.RUECK;
      JC    FChk;

      AN    #ZST.MicM1;  //neuer Befehl vor Ausgabe erst nochmal nach Hindernissen suchen
      S     #ZST.MicM1;
      JU    ErrA;

//----------------------------------
//prüfen ob Endziel erreicht
//----------------------------------
FChk: L     #End_Ziel_Inc;
      L     #ZST.PosInc;
      -D;
      DTR;
      ABS;
      RND;
      T     #Abstand;

      L     #Abstand;
      L     #PAR.Fahrt.Bereich_Pos;
      >D;
      ON    #IN.Pos_ok;
      A(;
      A     #ZST.Auto;
      O     #ZST.Semi;
      A     #ZST.SoftStop;
      );
      JC    ErrA;

      A     #ZST.Auto;
      O     #ZST.Semi;
      A(;
      A     #TMP.HW_akt_li;
      O     #TMP.HW_akt_re;
      );
      JC    HWe;
      S     #ZST.next_Step;
      R     #ZST.RUECKWAERTS_AKT;
      R     #ZST.VORWAERTS_AKT;

      SET;
      R     #TMP.old_vor_hoch;
      R     #TMP.old_rueck_runter;
      JU    ErrA;

HWe:  AN    #ZST.HW_mittig;
      JC    ErrA;
      JU    HW;


NETWORK
TITLE = Hubvorgang
Hub_Mig:NOP   0;
//------------------------------------
//Hubvorgang
//------------------------------------
      SET;
      R     #OUT.no_Brms;

      L     0;
      L     #TMP.HubZielInc_li;
      ==D;
      S     #MLD.Alarm_SW.ProgErr;  //Zielinkrement == 0 unzulässig

      L     #ZST.HubInc_li;
      -D;
      DTR;
      ABS;
      RND;
      T     #Abstand;
      L     #PAR.Hub.Bereich_Ziel;
      <=D;
      JC    brm_li;

      L     #TMP.HubZielInc_li;
      L     #ZST.HubInc_li;
      <D;
      S     #OUT.SENKEN_li;
      R     #OUT.HEBEN_li;
      >D;
      S     #OUT.HEBEN_li;
      R     #OUT.SENKEN_li;

//Geschwindigkeit langsam
brm_li:A     #lngsm_heb_li;
      A     #OUT.HEBEN_li;
      AN    #immer_schnell_li;
      O(;
      A     #lngsm_snk_li;
      A     #OUT.SENKEN_li;
      AN    #immer_schnell_li;
      );
      NOT;
      =     #OUT.HUB_EIL_li;

//Bremsvorgang
      L     #Abstand;
      L     #PAR.Hub.Bereich_Pos;
      <=D;
      A     #IN.Hub_ok_li;
      O(;
      AN    #IN.Anf_Hub_li;
      AN    #TMP.HW_akt_li;
      );
      =     #Hub_rdy_li;
      R     #OUT.HEBEN_li;
      R     #OUT.SENKEN_li;

      L     0;
      L     #HELP.HubZielInc_re;
      ==D;
      S     #MLD.Alarm_SW.ProgErr;  //Zielinkrement == 0 unzulässig

      L     #HELP.HubInc_re;
      -D;
      DTR;
      ABS;
      RND;
      T     #Abstand;
      L     #PAR.Hub.Bereich_Ziel;
      <=D;
      JC    brm_re;

      L     #HELP.HubZielInc_re;
      L     #HELP.HubInc_re;
      <D;
      S     #OUT.SENKEN_re;
      R     #OUT.HEBEN_re;
      >D;
      S     #OUT.HEBEN_re;
      R     #OUT.SENKEN_re;

//Geschwindigkeit langsam
brm_re:A     #lngsm_heb_re;
      A     #OUT.HEBEN_re;
      AN    #immer_schnell_re;
      O(;
      A     #lngsm_snk_re;
      A     #OUT.SENKEN_re;
      AN    #immer_schnell_re;
      );
      NOT;
      =     #OUT.HUB_EIL_re;

//Bremsvorgang
      L     #Abstand;
      L     #PAR.Hub.Bereich_Pos;
      <=D;
      A     #IN.Hub_ok_re;
      O(;
      AN    #IN.Anf_Hub_re;
      AN    #TMP.HW_akt_re;
      );
      =     #Hub_rdy_re;
      R     #OUT.HEBEN_re;
      R     #OUT.SENKEN_re;

// zur Sicherheit ,evtl.Langware am Haken
      A     #ZST.Hand;
      A     #ZST.Mittig;
      A     #OUT.SENKEN_li;
      A     #OUT.SENKEN_re;
      R     #OUT.HUB_EIL_li;
      R     #OUT.HUB_EIL_re;

      A     #OUT.HEBEN_li;
      O     #OUT.HEBEN_re;
      =     #OUT.HEBEN;
      =     #ZST.HEBEN_AKT;

      A     #OUT.SENKEN_li;
      O     #OUT.SENKEN_re;
      =     #OUT.SENKEN;
      =     #ZST.SENKEN_AKT;

      A     #Hub_rdy_li;
      A     #Hub_rdy_re;
      JC    HChk;
      JU    ErrA;

HChk: A     #TMP.HW_akt_li;  //HW aus Auto/Semi aufgerufen
      O     #TMP.HW_akt_re;
      R     #TMP.HW_akt_li;  //Positioniervorgang wird freigegeben.
      R     #TMP.HW_akt_re;
      JC    ErrA;
      S     #ZST.next_Step;  //Fertig
      SET;
      R     #TMP.old_vor_hoch;
      R     #TMP.old_rueck_runter;
      JU    ErrA;


NETWORK
TITLE = Fehlerbehandlung/Überwachungsfunktionen Hand/Auto
// überwacht die Fahrwagenfunktionen in den betriebsarten Hand und Auto
ErrA: NOP   0;
//-----------------------------
//WT am TW bei Endlage "unten"
//-----------------------------
      A     #WTon_li;
      A     #ZST.Unten_li;
      AN    #ZST.Mittig;
      A     #ZST.Auto;
      AN    #ZST.HEBEN_AKT;
      AN    #ZST.SENKEN_AKT;
      =     #MLD.Alarm_SW.WTon_bei_SU_li;

      A     #WTon_re;
      A     #ZST.Unten_re;
      AN    #ZST.Mittig;
      A     #ZST.Auto;
      AN    #ZST.HEBEN_AKT;
      AN    #ZST.SENKEN_AKT;
      =     #MLD.Alarm_SW.WTon_bei_SU_re;

//-----------------------------------
//Hubbewegung bei ignorierter Sperre
//-----------------------------------
      L     #Adr_IstPos;
      LAR1;
      A     #OUT.SENKEN_li;
      OPN   "DB_POS";
      A     DBX [AR1, P#10.3];  //Freigabe Einfahrsperre ignor.
      A     DBX [AR1, P#9.1];  //Einfahrsperre Freigabe
      R     #OUT.SENKEN_li;

      A     #OUT.SENKEN_re;
      OPN   "DB_POS";
      A     DBX [AR1, P#110.3];  //Freigabe Einfahrsperre ignor.
      A     DBX [AR1, P#109.1];  //Einfahrsperre Freigabe
      R     #OUT.SENKEN_re;

//--------------------------
//Befehl wird nicht ausgeführt
//--------------------------
      A     #ZST.HEBEN_AKT;
      O     #ZST.SENKEN_AKT;
      O     #ZST.VORWAERTS_AKT;
      O     #ZST.RUECKWAERTS_AKT;
      AN    #OUT.HEBEN_li;
      AN    #OUT.HEBEN_re;
      AN    #OUT.SENKEN_li;
      AN    #OUT.SENKEN_re;
      AN    #OUT.VOR;
      AN    #OUT.RUECK;
      AN    #ZST.FEHLER;
      JC    ck35;
      R     #C1_rdy;

      L     1800;  //entspricht 3min
      T     #TMP.count1;

ck35: A     #C1_rdy;
      S     #MLD.Alarm_SW.TO_Befehl;

//---------------------------------------------
//Hubbewegung nicht erlaubt (HCA: unverzögert)
//---------------------------------------------
      L     #Adr_IstPos;
      LAR1;
      A     #OUT.HEBEN_li;
      O     #OUT.SENKEN_li;
      OPN   "DB_POS";
      A     DBX [AR1, P#7.3];  //Hubbewegung nicht erlaubt
      R     #OUT.HEBEN_li;
      R     #OUT.SENKEN_li;
      S     #MLD.Alarm_SW.Hub_nen_li;

      L     #Adr_IstPos;
      LAR1;
      A     #OUT.HEBEN_re;
      O     #OUT.SENKEN_re;
      OPN   "DB_POS";
      A     DBX [AR1, P#107.3];  //Hubbewegung nicht erlaubt
      R     #OUT.HEBEN_re;
      R     #OUT.SENKEN_re;
      S     #MLD.Alarm_SW.Hub_nen_re;

//--------------------------
//Timeout Heben
//--------------------------

      AN    #OUT.HUB_EIL_li;
      A     #OUT.SENKEN_li;
      JC    lngs_li;
      AN    #OUT.HUB_EIL_li;
      A     #OUT.HEBEN_li;
      JC    lngs_li;
      L     #PAR.Hub.TO_Heben_Senken_hi;
      T     #TO_Hub;
      JU    THUB_li;
lngs_li:L     #PAR.Hub.TO_Heben_Senken_low;
      T     #TO_Hub;

THUB_li:L     #ZST.HubInc_li;
      L     #TMP.AltHub_li;
      -D;
      DTR;
      ABS;
      RND;
      L     #PAR.Hub.delta_s;
      <=D;
      =     #noMove;
      JC    TOH_li;
      L     #ZST.HubInc_li;
      T     #TMP.AltHub_li;

TOH_li:A     #OUT.HEBEN_li;
      O     #OUT.SENKEN_li;
      AN    #ZST.Halt;
      A     #noMove;
      AN(;
      A     #OUT.SENKEN_li;
      A     #TMP.old_vor_hoch;
      O;
      A     #OUT.HEBEN_li;
      A     #TMP.old_rueck_runter;
      );
      L     #TO_Hub;
      SD    T [#Timer2];

      A     T [#Timer2];
      S     #MLD.Alarm_SW.TO_Hub_li;

      AN    #OUT.HUB_EIL_re;
      A     #OUT.SENKEN_re;
      JC    lngs_re;
      AN    #OUT.HUB_EIL_re;
      A     #OUT.HEBEN_re;
      JC    lngs_re;
      L     #PAR.Hub.TO_Heben_Senken_hi;
      T     #TO_Hub;
      JU    THUB_re;
lngs_re:L     #PAR.Hub.TO_Heben_Senken_low;
      T     #TO_Hub;

THUB_re:L     #HELP.HubInc_re;
      L     #HELP.AltHub_re;
      -D;
      DTR;
      ABS;
      RND;
      L     #PAR.Hub.delta_s;
      <=D;
      =     #noMove;
      JC    TOH_re;
      L     #HELP.HubInc_re;
      T     #HELP.AltHub_re;

TOH_re:A     #OUT.HEBEN_re;
      O     #OUT.SENKEN_re;
      AN    #ZST.Halt;
      A     #noMove;
      AN(;
      A     #OUT.SENKEN_re;
      A     #TMP.old_vor_hoch;
      O;
      A     #OUT.HEBEN_re;
      A     #TMP.old_rueck_runter;
      );
      L     #TO_Hub;
      SD    T [#Timer8];

      A     T [#Timer8];
      S     #MLD.Alarm_SW.TO_Hub_re;

//--------------------------
//Timeout Fahren
//--------------------------
      L     #ZST.PosInc;
      L     #TMP.AltPos;
      -D;
      DTR;
      ABS;
      RND;
      L     #PAR.Fahrt.delta_s;
      <=D;
      =     #noMove;
      JC    TOF;
      L     #ZST.PosInc;
      T     #TMP.AltPos;

TOF:  A     #OUT.VOR;
      O     #OUT.RUECK;
      AN    #ZST.Halt;
      A     #noMove;
      L     #PAR.Fahrt.TO_Fahren;
      SD    T [#Timer1];

      L     #Abstand;
      L     #PAR.Fahrt.Bereich_Pos;
      <=D;
      A     T [#Timer1];
      R     #OUT.VOR;
      R     #OUT.RUECK;
      >D;
      A     T [#Timer1];
      S     #MLD.Alarm_SW.TO_Fahrt;
//--------------------------
//HEBEN POS-NICHT BELEGT?
//--------------------------
      L     #Adr_IstPos;
      LAR1;
      OPN   "DB_POS";
      AN    DBX [AR1, P#96.0];  //belegt
      A     #ZST.Auto;
      AN    #ZST.HW_mittig;
      AN    #ZST.Ofs_mittig;
      A     #ZST.low_SU_li;
      A     #OUT.HEBEN_li;
      S     #MLD.Alarm_SW.Heben_WT_li;

      AN    DBX [AR1, P#196.0];  //belegt
      A     #ZST.Auto;
      AN    #ZST.HW_mittig;
      AN    #ZST.Ofs_mittig;
      A     #ZST.low_SU_re;
      A     #OUT.HEBEN_re;
      S     #MLD.Alarm_SW.Heben_WT_re;

//--------------------------
//SENKEN POS-BELEGT?
//--------------------------
      L     1800;  // Gemessen mit Hr. Pahl, höchster Wasserstand wenn Becken voll + voll belegt #PAR.Hub.Ebene1
      L     #ZST.HubInc_li;
      <D;
      A     #OUT.SENKEN_li;
      A     #ZST.Mittig;
      A(;
      L     #ZST.POSITION_li;
      L     23;
      <=I;
      );
      =     #Freigabe;

      L     #HELP.AW_Summe_WZ_li;
      L     #HELP.Summe_WZ_li;
      -R;
      L     75.0;  //50.0
      >R;
      A     #Freigabe;
      =     #ErrIn.Alarm.POS_BELEGT_li;

      L     #Adr_IstPos;
      LAR1;
      OPN   "DB_POS";
      L     DBB [AR1, P#35.0];  //WT-DB
      L     0;
      <>I;
      O     DBX [AR1, P#96.0];  //belegt
      A     #OUT.SENKEN_li;
      AN    #ZST.HW_mittig;
      AN    #ZST.Ofs_mittig;
      A     #ZST.HubSensor_li;
      O     #ErrIn.Alarm.POS_BELEGT_li;
      AN    #ZST.low_SU_li;
      S     #MLD.Alarm_SW.Senken_WT_li;

      L     1800;  // Gemessen mit Hr. Pahl, höchster Wasserstand wenn Becken voll + voll belegt #PAR.Hub.Ebene1
      L     #HELP.HubInc_re;
      <D;
      A     #OUT.SENKEN_re;
      A     #ZST.Mittig;
      A(;
      L     #ZST.POSITION_re;
      L     24;
      <=I;
      );
      =     #Freigabe;

      L     #HELP.AW_Summe_WZ_re;
      L     #HELP.Summe_WZ_re;
      -R;
      L     75.0;  //50.0
      >R;
      A     #Freigabe;
      =     #ErrIn.Alarm.POS_BELEGT_re;

      L     #Adr_IstPos;
      LAR1;
      OPN   "DB_POS";
      L     DBB [AR1, P#135.0];  //WT-DB
      L     0;
      <>I;
      O     DBX [AR1, P#196.0];  //belegt
      A     #OUT.SENKEN_re;
      AN    #ZST.HW_mittig;
      AN    #ZST.Ofs_mittig;
      A     #ZST.HubSensor_re;
      O     #ErrIn.Alarm.POS_BELEGT_re;
      AN    #ZST.low_SU_re;
      S     #MLD.Alarm_SW.Senken_WT_re;

//--------------------------
//Senken trotz gesperrt
//--------------------------
      OPN   "DB_POS";
      A     DBX [AR1, P#9.1];  //Einfahrsperre Freigabe
      AN    DBX [AR1, P#10.3];  //Einfahrsperre Freigabe ignor.
      O     DBX [AR1, P#7.0];  //Einfahrsperrre
      O(;  // 2024-08
      L     #ZST.POSITION_li;
      L     13;
      <I;
      A     #WT_151_li;
      );
      O(;
      L     11;
      L     #ZST.POSITION_li;
      <I;
      A(;
      L     25;
      <I;
      );
      A     #WT_161_li;
      );
      A     #OUT.SENKEN_li;
      AN    #ZST.HW_mittig;
      AN    #ZST.Ofs_mittig;
      A     #ZST.HubSensor_li;
      AN    #ZST.low_SU_li;
      S     #MLD.Alarm_SW.Senken_Sperre_li;

      OPN   "DB_POS";
      A     DBX [AR1, P#109.1];  //Einfahrsperre Freigabe
      AN    DBX [AR1, P#110.3];  //Einfahrsperre Freigabe ignor.
      O     DBX [AR1, P#107.0];  //Einfahrsperrre
      O(;  // 2024-08
      L     #ZST.POSITION_re;
      L     14;
      <I;
      A     #WT_151_re;
      );
      O(;
      L     12;
      L     #ZST.POSITION_re;
      <I;
      A(;
      L     26;
      <I;
      );
      A     #WT_161_re;
      );
      A     #OUT.SENKEN_re;
      AN    #ZST.HW_mittig;
      AN    #ZST.Ofs_mittig;
      A     #ZST.HubSensor_re;
      AN    #ZST.low_SU_re;
      S     #MLD.Alarm_SW.Senken_Sperre_re;

//--------------------------
//Senken in falschen BadTyp
//--------------------------
      SET;
      R     #MLD.Alarm_SW.PosTyp_WT_Typ_li;

      L     #Adr_IstPos;
      LAR1;
      OPN   "DB_POS";
      L     DBB [AR1, P#11.0];  //"DB_POS".POS[0].Detailtyp
      T     #Pos_WT_Typ;

      L     #WT_Typ_li;  //Hi-Nibble prüfen vom WT
      AW    16#00F0;
      JZ    hok_li;

      L     #Pos_WT_Typ;
      AW    16#00F0;
      JZ    hok_li;
      <>I;
      A     #OUT.SENKEN_li;
      S     #MLD.Alarm_SW.PosTyp_WT_Typ_li;
      JC    E_ok_li;

hok_li:AN    #Typ_chk;
      JC    E_ok_li;

      L     #WT_Typ_li;  //Lo-Nibble prüfen vom WT
      AW    16#000F;
      JZ    E_ok_li;

      L     #Pos_WT_Typ;
      AW    16#000F;
      JZ    E_ok_li;
      <>I;
      A     #OUT.SENKEN_li;
      S     #MLD.Alarm_SW.PosTyp_WT_Typ_li;

E_ok_li:NOP   0;

      SET;
      R     #MLD.Alarm_SW.PosTyp_WT_Typ_re;

      L     #Adr_IstPos;
      LAR1;
      OPN   "DB_POS";
      L     DBB [AR1, P#11.0];  //"DB_POS".POS[0].Detailtyp
      T     #Pos_WT_Typ;

      L     #WT_Typ_re;  //Hi-Nibble prüfen vom WT
      AW    16#00F0;
      JZ    hok_re;

      L     #Pos_WT_Typ;
      AW    16#00F0;
      JZ    hok_re;
      <>I;
      A     #OUT.SENKEN_re;
      S     #MLD.Alarm_SW.PosTyp_WT_Typ_re;
      JC    E_ok_re;

hok_re:AN    #Typ_chk;
      JC    E_ok_re;

      L     #WT_Typ_re;  //Lo-Nibble prüfen vom WT
      AW    16#000F;
      JZ    E_ok_re;

      L     #Pos_WT_Typ;
      AW    16#000F;
      JZ    E_ok_re;
      <>I;
      A     #OUT.SENKEN_re;
      S     #MLD.Alarm_SW.PosTyp_WT_Typ_re;

E_ok_re:NOP   0;

//--------------------------
//WARENFAHRT SO-TESTEN
//--------------------------
      A     #OUT.VOR;
      O     #OUT.RUECK;
      A(;
      A     #WTon_li;
      AN    #ZST.Oben_li;
      A     #ZST.Auto;
      O;
      A     #WTon_li;
      AN    #ZST.Unten_li;
      AN    #ZST.Oben_li;
      );
      AN    #ErrIn.Alarm.Profinet_IO_nok;
      S     #MLD.Alarm_SW.SO_fehlt_li;

      A     #OUT.VOR;
      O     #OUT.RUECK;
      A(;
      A     #WTon_re;
      AN    #ZST.Oben_re;
      A     #ZST.Auto;
      O;
      A     #WTon_re;
      AN    #ZST.Unten_re;
      AN    #ZST.Oben_re;
      );
      AN    #ErrIn.Alarm.Profinet_IO_nok;
      S     #MLD.Alarm_SW.SO_fehlt_re;

//--------------------------
//LEERFAHRT SU-TESTEN
//--------------------------
      A     #OUT.VOR;
      O     #OUT.RUECK;
      A(;
      AN    #WTon_li;
      AN    #ZST.Unten_li;
      A     #ZST.Auto;
      O;
      AN    #WTon_li;
      AN    #ZST.Unten_li;
      AN    #ZST.Oben_li;
      );
      AN    #ErrIn.Alarm.Profinet_IO_nok;
      S     #MLD.Alarm_SW.SU_fehlt_li;

      A     #OUT.VOR;
      O     #OUT.RUECK;
      A(;
      AN    #WTon_re;
      AN    #ZST.Unten_re;
      A     #ZST.Auto;
      O;
      AN    #WTon_re;
      AN    #ZST.Unten_re;
      AN    #ZST.Oben_re;
      );
      AN    #ErrIn.Alarm.Profinet_IO_nok;
      S     #MLD.Alarm_SW.SU_fehlt_re;

//-------------------------------
//HUBBEWEGUNG IN MITTENPOSITION?
//-------------------------------
      A     #OUT.HEBEN_li;
      O     #OUT.SENKEN_li;
      AN    #ZST.Mittig;
      AN(;
      A     #ZST.HW_mittig;
      O     #ZST.Ofs_mittig;
      AN    #WTon_li;
      );
      S     #MLD.Alarm_SW.Hub_not_mittig_li;

      A     #OUT.HEBEN_re;
      O     #OUT.SENKEN_re;
      AN    #ZST.Mittig;
      AN(;
      A     #ZST.HW_mittig;
      O     #ZST.Ofs_mittig;
      AN    #WTon_re;
      );
      S     #MLD.Alarm_SW.Hub_not_mittig_re;

//-------------------------------
// Überwachung Wägezellen
//-------------------------------
//links
      L     #HELP.WZ_links_1;
      L     #HELP.WZ_links_2;
      +R;
      T     #HELP.Sum_WZ_li_vorn;
      L     #HELP.AW_WZ_li_vorn;
      -R;
      ABS;
      L     #HELP.Tol_UeW_WZ;
      >R;
      A     #OUT.VOR;
      =     #Kollision;

      L     #HELP.WZ_links_3;
      L     #HELP.WZ_links_4;
      +R;
      T     #HELP.Sum_WZ_li_hinten;
      L     #HELP.AW_WZ_li_hinten;
      -R;
      ABS;
      L     #HELP.Tol_UeW_WZ;
      >R;
      A     #OUT.RUECK;
      S     #Kollision;

      A     #Kollision;
      A     #ZST.Unten_li;
      =     #ErrIn.Alarm.Koll_LF;

      A     #Kollision;
      A     #ZST.Oben_li;
      =     #ErrIn.Alarm.Koll_WF;
//rechts
      L     #HELP.WZ_rechts_1;
      L     #HELP.WZ_rechts_2;
      +R;
      T     #HELP.Sum_WZ_re_vorn;
      L     #HELP.AW_WZ_re_vorn;
      -R;
      ABS;
      L     #HELP.Tol_UeW_WZ;
      >R;
      A     #OUT.VOR;
      =     #Kollision;

